LIN {X 0,Y 417.016,Z 627.534,A -85,B 0,C 180,E1 -10173.865,E2 -10173.865} C_VEL
LIN {X 0,Y 417.122,Z 624.59,A -85,B 0,C 180,E1 -10175.317,E2 -10175.317} C_VEL
LIN {X 0,Y 417.232,Z 620.603,A -85,B 0,C 180,E1 -10176.771,E2 -10176.771} C_VEL
LIN {X 0,Y 417.503,Z 614.475,A -85,B 0,C 180,E1 -10178.47,E2 -10178.47} C_VEL
LIN {X 0,Y 417.901,Z 607.782,A -85,B 0,C 180,E1 -10179.926,E2 -10179.926} C_VEL
LIN {X 0,Y 418.469,Z 599.483,A -85,B 0,C 180,E1 -10181.381,E2 -10181.381} C_VEL
LIN {X 0,Y 419.119,Z 590.981,A -85,B 0,C 180,E1 -10182.591,E2 -10182.591} C_VEL
LIN {X 0,Y 419.778,Z 581.378,A -85,B 0,C 180,E1 -10183.708,E2 -10183.708} C_VEL
LIN {X 0,Y 420.547,Z 570.086,A -85,B 0,C 180,E1 -10184.764,E2 -10184.764} C_VEL
LIN {X 0,Y 421.293,Z 558.7,A -85,B 0,C 180,E1 -10185.604,E2 -10185.604} C_VEL
LIN {X 0,Y 421.95,Z 547.015,A -85,B 0,C 180,E1 -10186.262,E2 -10186.262} C_VEL
LIN {X 0,Y 422.541,Z 534.469,A -85,B 0,C 180,E1 -10186.766,E2 -10186.766} C_VEL
LIN {X 0,Y 422.903,Z 521.748,A -85,B 0,C 180,E1 -10187.094,E2 -10187.094} C_VEL
LIN {X 0,Y 423.634,Z 443.257,A -85,B 0,C 180,E1 -10188.435,E2 -10188.435} C_VEL
LIN {X 0,Y 419.657,Z 417.924,A -85,B 0,C 180,E1 -10189.065,E2 -10189.065} C_VEL
LIN {X 0,Y 420.847,Z 399.93,A -85,B 0,C 180,E1 -10192.587,E2 -10192.587} C_VEL
LIN {X 0,Y 421.466,Z 390.877,A -85,B 0,C 180,E1 -10194.375,E2 -10194.375} C_VEL
LIN {X 0,Y 419.594,Z 380.403,A -85,B 0,C 180,E1 -10196.618,E2 -10196.618} C_VEL
LIN {X 0,Y 418.306,Z 374.38,A -85,B 0,C 180,E1 -10198.004,E2 -10198.004} C_VEL
LIN {X 0,Y 418.211,Z 374.394,A -85,B 0,C 180,E1 -10201.395,E2 -10201.395} C_VEL
LIN {X 0,Y 418.264,Z 374.38,A -85,B 0,C 180,E1 -10204.58,E2 -10204.58} C_VEL
LIN {X 0,Y 418.233,Z 374.389,A -85,B 0,C 180,E1 -10207.834,E2 -10207.834} C_VEL
LIN {X 0,Y 418.258,Z 374.382,A -85,B 0,C 180,E1 -10210.943,E2 -10210.943} C_VEL
LIN {X 0,Y 418.214,Z 374.392,A -85,B 0,C 180,E1 -10213.73,E2 -10213.73} C_VEL
LIN {X 0,Y 418.264,Z 374.38,A -85,B 0,C 180,E1 -10216.456,E2 -10216.456} C_VEL
LIN {X 0,Y 418.263,Z 374.383,A -85,B 0,C 180,E1 -10219.122,E2 -10219.122} C_VEL
LIN {X 0,Y 418.233,Z 374.385,A -85,B 0,C 180,E1 -10222.164,E2 -10222.164} C_VEL
LIN {X 0,Y 418.26,Z 374.388,A -85,B 0,C 180,E1 -10225.419,E2 -10225.419} C_VEL
LIN {X 0,Y 418.21,Z 374.387,A -85,B 0,C 180,E1 -10228.604,E2 -10228.604} C_VEL
LIN {X 0,Y 418.289,Z 374.378,A -85,B 0,C 180,E1 -10231.936,E2 -10231.936} C_VEL
LIN {X 0,Y 418.283,Z 374.384,A -85,B 0,C 180,E1 -10235.162,E2 -10235.162} C_VEL
LIN {X 0,Y 418.228,Z 374.385,A -85,B 0,C 180,E1 -10238.303,E2 -10238.303} C_VEL
LIN {X 0,Y 418.276,Z 374.384,A -85,B 0,C 180,E1 -10241.383,E2 -10241.383} C_VEL
LIN {X 0,Y 418.294,Z 374.377,A -85,B 0,C 180,E1 -10244.406,E2 -10244.406} C_VEL
LIN {X 0,Y 418.362,Z 374.372,A -85,B 0,C 180,E1 -10247.386,E2 -10247.386} C_VEL
LIN {X 0,Y 418.353,Z 374.369,A -85,B 0,C 180,E1 -10250.329,E2 -10250.329} C_VEL
LIN {X 0,Y 418.485,Z 374.357,A -85,B 0,C 180,E1 -10253.249,E2 -10253.249} C_VEL
LIN {X 0,Y 418.335,Z 374.376,A -85,B 0,C 180,E1 -10255.182,E2 -10255.182} C_VEL
LIN {X 0,Y 418.537,Z 374.346,A -85,B 0,C 180,E1 -10258.075,E2 -10258.075} C_VEL
LIN {X 0,Y 418.666,Z 374.33,A -85,B 0,C 180,E1 -10260,E2 -10260} C_VEL
LIN {X 0,Y 418.504,Z 374.358,A -85,B 0,C 180,E1 -10262.888,E2 -10262.888} C_VEL
LIN {X 0,Y 418.486,Z 374.359,A -85,B 0,C 180,E1 -10266.751,E2 -10266.751} C_VEL
LIN {X 0,Y 418.352,Z 374.369,A -85,B 0,C 180,E1 -10269.671,E2 -10269.671} C_VEL
LIN {X 0,Y 418.347,Z 374.374,A -85,B 0,C 180,E1 -10273.007,E2 -10273.007} C_VEL
LIN {X 0,Y 418.305,Z 374.382,A -85,B 0,C 180,E1 -10276.736,E2 -10276.736} C_VEL
LIN {X 0,Y 418.264,Z 374.38,A -85,B 0,C 180,E1 -10279.791,E2 -10279.791} C_VEL
LIN {X 0,Y 418.231,Z 374.39,A -85,B 0,C 180,E1 -10282.737,E2 -10282.737} C_VEL
LIN {X 0,Y 418.264,Z 374.381,A -85,B 0,C 180,E1 -10285.905,E2 -10285.905} C_VEL
LIN {X 0,Y 418.258,Z 374.382,A -85,B 0,C 180,E1 -10289.163,E2 -10289.163} C_VEL
LIN {X 0,Y 418.252,Z 374.385,A -85,B 0,C 180,E1 -10292.845,E2 -10292.845} C_VEL
LIN {X 0,Y 418.243,Z 374.387,A -85,B 0,C 180,E1 -10296.239,E2 -10296.239} C_VEL
LIN {X 0,Y 418.26,Z 374.381,A -85,B 0,C 180,E1 -10299.681,E2 -10299.681} C_VEL
LIN {X 0,Y 418.282,Z 374.385,A -85,B 0,C 180,E1 -10302.33,E2 -10302.33} C_VEL
LIN {X 0,Y 418.248,Z 374.382,A -85,B 0,C 180,E1 -10305.112,E2 -10305.112} C_VEL
LIN {X 0,Y 418.238,Z 374.385,A -85,B 0,C 180,E1 -10307.768,E2 -10307.768} C_VEL
LIN {X 0,Y 418.258,Z 374.384,A -85,B 0,C 180,E1 -10310.619,E2 -10310.619} C_VEL
LIN {X 0,Y 418.245,Z 374.387,A -85,B 0,C 180,E1 -10313.977,E2 -10313.977} C_VEL
LIN {X 0,Y 418.257,Z 374.381,A -85,B 0,C 180,E1 -10317.157,E2 -10317.157} C_VEL
LIN {X 0,Y 418.269,Z 374.38,A -85,B 0,C 180,E1 -10320.896,E2 -10320.896} C_VEL
LIN {X 0,Y 418.269,Z 374.387,A -85,B 0,C 180,E1 -10324.096,E2 -10324.096} C_VEL
LIN {X 0,Y 418.25,Z 374.479,A -85,B 0,C 180,E1 -10327.293,E2 -10327.293} C_VEL
LIN {X 0,Y 419.963,Z 383.206,A -85,B 0,C 180,E1 -10329.579,E2 -10329.579} C_VEL
LIN {X 0,Y 420.227,Z 386.742,A -85,B 0,C 180,E1 -10330.459,E2 -10330.459} C_VEL
LIN {X 0,Y 420.053,Z 389.099,A -85,B 0,C 180,E1 -10331.02,E2 -10331.02} C_VEL
LIN {X 0,Y 424.09,Z 408.927,A -85,B 0,C 180,E1 -10331.56,E2 -10331.56} C_VEL
LIN {X 0,Y 423.113,Z 496.309,A -85,B 0,C 180,E1 -10333.071,E2 -10333.071} C_VEL
LIN {X 0,Y 422.612,Z 510.138,A -85,B 0,C 180,E1 -10333.516,E2 -10333.516} C_VEL
LIN {X 0,Y 422.063,Z 522.517,A -85,B 0,C 180,E1 -10334.115,E2 -10334.115} C_VEL
LIN {X 0,Y 421.498,Z 534.349,A -85,B 0,C 180,E1 -10334.899,E2 -10334.899} C_VEL
LIN {X 0,Y 420.864,Z 544.797,A -85,B 0,C 180,E1 -10335.778,E2 -10335.778} C_VEL
LIN {X 0,Y 420.185,Z 554.863,A -85,B 0,C 180,E1 -10336.827,E2 -10336.827} C_VEL
LIN {X 0,Y 419.491,Z 563.403,A -85,B 0,C 180,E1 -10337.912,E2 -10337.912} C_VEL
LIN {X 0,Y 418.903,Z 571.264,A -85,B 0,C 180,E1 -10339.121,E2 -10339.121} C_VEL
LIN {X 0,Y 418.314,Z 578.947,A -85,B 0,C 180,E1 -10340.572,E2 -10340.572} C_VEL
LIN {X 0,Y 417.789,Z 585.995,A -85,B 0,C 180,E1 -10342.266,E2 -10342.266} C_VEL
LIN {X 0,Y 417.601,Z 589.304,A -85,B 0,C 180,E1 -10343.245,E2 -10343.245} C_VEL
LIN {X 0,Y 416.888,Z 591.511,A -85,B 0,C 180,E1 -10343.994,E2 -10343.994} C_VEL
LIN {X 0,Y 413.901,Z 594.609,A -85,B 0,C 180,E1 -10345.222,E2 -10345.222} C_VEL
LIN {X 0,Y 411.354,Z 596.611,A -85,B 0,C 180,E1 -10346.233,E2 -10346.233} C_VEL
LIN {X 0,Y 410.212,Z 597.769,A -85,B 0,C 180,E1 -10347.029,E2 -10347.029} C_VEL
LIN {X 0,Y 410.095,Z 598.052,A -85,B 0,C 180,E1 -10347.302,E2 -10347.302} C_VEL
LIN {X 0,Y 409.96,Z 599.41,A -85,B 0,C 180,E1 -10349.018,E2 -10349.018} C_VEL
LIN {X 0,Y 409.949,Z 599.643,A -85,B 0,C 180,E1 -10350,E2 -10350} C_VEL
LIN {X 0,Y 409.96,Z 599.455,A -85,B 0,C 180,E1 -10350.982,E2 -10350.982} C_VEL
LIN {X 0,Y 410.131,Z 597.905,A -85,B 0,C 180,E1 -10352.947,E2 -10352.947} C_VEL
LIN {X 0,Y 410.122,Z 596.556,A -85,B 0,C 180,E1 -10353.93,E2 -10353.93} C_VEL
LIN {X 0,Y 410.301,Z 593.697,A -85,B 0,C 180,E1 -10355.406,E2 -10355.406} C_VEL
LIN {X 0,Y 410.543,Z 589.82,A -85,B 0,C 180,E1 -10356.882,E2 -10356.882} C_VEL
LIN {X 0,Y 410.856,Z 584.818,A -85,B 0,C 180,E1 -10358.36,E2 -10358.36} C_VEL
LIN {X 0,Y 411.393,Z 578.516,A -85,B 0,C 180,E1 -10359.836,E2 -10359.836} C_VEL
LIN {X 0,Y 412.034,Z 570.627,A -85,B 0,C 180,E1 -10361.312,E2 -10361.312} C_VEL
LIN {X 0,Y 412.639,Z 562.584,A -85,B 0,C 180,E1 -10362.542,E2 -10362.542} C_VEL
LIN {X 0,Y 413.512,Z 552.76,A -85,B 0,C 180,E1 -10363.765,E2 -10363.765} C_VEL
LIN {X 0,Y 414.125,Z 543.099,A -85,B 0,C 180,E1 -10364.747,E2 -10364.747} C_VEL
LIN {X 0,Y 414.814,Z 532.639,A -85,B 0,C 180,E1 -10365.602,E2 -10365.602} C_VEL
LIN {X 0,Y 415.467,Z 520.04,A -85,B 0,C 180,E1 -10366.396,E2 -10366.396} C_VEL
LIN {X 0,Y 416.011,Z 507.426,A -85,B 0,C 180,E1 -10366.974,E2 -10366.974} C_VEL
LIN {X 0,Y 416.372,Z 495.481,A -85,B 0,C 180,E1 -10367.338,E2 -10367.338} C_VEL
LIN {X 0,Y 417.31,Z 409.13,A -85,B 0,C 180,E1 -10368.85,E2 -10368.85} C_VEL
LIN {X 0,Y 413.176,Z 389.255,A -85,B 0,C 180,E1 -10369.436,E2 -10369.436} C_VEL
LIN {X 0,Y 413.003,Z 384.502,A -85,B 0,C 180,E1 -10370.621,E2 -10370.621} C_VEL
LIN {X 0,Y 411.231,Z 375.268,A -85,B 0,C 180,E1 -10373.11,E2 -10373.11} C_VEL
LIN {X 0,Y 411.239,Z 375.258,A -85,B 0,C 180,E1 -10376.38,E2 -10376.38} C_VEL
LIN {X 0,Y 411.2,Z 375.264,A -85,B 0,C 180,E1 -10379.712,E2 -10379.712} C_VEL
LIN {X 0,Y 411.206,Z 375.26,A -85,B 0,C 180,E1 -10383.155,E2 -10383.155} C_VEL
LIN {X 0,Y 411.194,Z 375.261,A -85,B 0,C 180,E1 -10386.552,E2 -10386.552} C_VEL
LIN {X 0,Y 411.216,Z 375.264,A -85,B 0,C 180,E1 -10389.728,E2 -10389.728} C_VEL
LIN {X 0,Y 411.171,Z 375.265,A -85,B 0,C 180,E1 -10393.133,E2 -10393.133} C_VEL
LIN {X 0,Y 411.224,Z 375.263,A -85,B 0,C 180,E1 -10395.872,E2 -10395.872} C_VEL
LIN {X 0,Y 411.206,Z 375.259,A -85,B 0,C 180,E1 -10398.763,E2 -10398.763} C_VEL
LIN {X 0,Y 411.199,Z 375.263,A -85,B 0,C 180,E1 -10402.027,E2 -10402.027} C_VEL
LIN {X 0,Y 411.201,Z 375.266,A -85,B 0,C 180,E1 -10405.666,E2 -10405.666} C_VEL
LIN {X 0,Y 411.183,Z 375.265,A -85,B 0,C 180,E1 -10409.152,E2 -10409.152} C_VEL
LIN {X 0,Y 411.252,Z 375.253,A -85,B 0,C 180,E1 -10412.522,E2 -10412.522} C_VEL
LIN {X 0,Y 411.221,Z 375.261,A -85,B 0,C 180,E1 -10415.784,E2 -10415.784} C_VEL
LIN {X 0,Y 411.191,Z 375.264,A -85,B 0,C 180,E1 -10418.965,E2 -10418.965} C_VEL
LIN {X 0,Y 411.245,Z 375.255,A -85,B 0,C 180,E1 -10422.084,E2 -10422.084} C_VEL
LIN {X 0,Y 411.255,Z 375.258,A -85,B 0,C 180,E1 -10425.147,E2 -10425.147} C_VEL
LIN {X 0,Y 411.291,Z 375.249,A -85,B 0,C 180,E1 -10428.167,E2 -10428.167} C_VEL
LIN {X 0,Y 411.474,Z 375.226,A -85,B 0,C 180,E1 -10432.146,E2 -10432.146} C_VEL
LIN {X 0,Y 411.467,Z 375.227,A -85,B 0,C 180,E1 -10434.118,E2 -10434.118} C_VEL
LIN {X 0,Y 411.506,Z 375.222,A -85,B 0,C 180,E1 -10438.042,E2 -10438.042} C_VEL
LIN {X 0,Y 411.635,Z 375.206,A -85,B 0,C 180,E1 -10440,E2 -10440} C_VEL
LIN {X 0,Y 411.46,Z 375.233,A -85,B 0,C 180,E1 -10442.937,E2 -10442.937} C_VEL
LIN {X 0,Y 411.453,Z 375.234,A -85,B 0,C 180,E1 -10446.867,E2 -10446.867} C_VEL
LIN {X 0,Y 411.301,Z 375.247,A -85,B 0,C 180,E1 -10449.839,E2 -10449.839} C_VEL
LIN {X 0,Y 411.305,Z 375.252,A -85,B 0,C 180,E1 -10453.109,E2 -10453.109} C_VEL
LIN {X 0,Y 411.249,Z 375.261,A -85,B 0,C 180,E1 -10456.889,E2 -10456.889} C_VEL
LIN {X 0,Y 411.223,Z 375.257,A -85,B 0,C 180,E1 -10459.987,E2 -10459.987} C_VEL
LIN {X 0,Y 411.196,Z 375.263,A -85,B 0,C 180,E1 -10463.148,E2 -10463.148} C_VEL
LIN {X 0,Y 411.231,Z 375.259,A -85,B 0,C 180,E1 -10466.381,E2 -10466.381} C_VEL
LIN {X 0,Y 411.194,Z 375.261,A -85,B 0,C 180,E1 -10469.713,E2 -10469.713} C_VEL
LIN {X 0,Y 411.2,Z 375.262,A -85,B 0,C 180,E1 -10473.156,E2 -10473.156} C_VEL
LIN {X 0,Y 411.19,Z 375.268,A -85,B 0,C 180,E1 -10476.554,E2 -10476.554} C_VEL
LIN {X 0,Y 411.223,Z 375.257,A -85,B 0,C 180,E1 -10479.731,E2 -10479.731} C_VEL
LIN {X 0,Y 411.218,Z 375.259,A -85,B 0,C 180,E1 -10483.128,E2 -10483.128} C_VEL
LIN {X 0,Y 411.173,Z 375.265,A -85,B 0,C 180,E1 -10485.88,E2 -10485.88} C_VEL
LIN {X 0,Y 411.203,Z 375.26,A -85,B 0,C 180,E1 -10489.5,E2 -10489.5} C_VEL
LIN {X 0,Y 411.199,Z 375.263,A -85,B 0,C 180,E1 -10492.028,E2 -10492.028} C_VEL
LIN {X 0,Y 411.205,Z 375.26,A -85,B 0,C 180,E1 -10495.667,E2 -10495.667} C_VEL
LIN {X 0,Y 411.19,Z 375.264,A -85,B 0,C 180,E1 -10499.153,E2 -10499.153} C_VEL
LIN {X 0,Y 411.253,Z 375.293,A -85,B 0,C 180,E1 -10501.762,E2 -10501.762} C_VEL
LIN {X 0,Y 413.552,Z 386.393,A -85,B 0,C 180,E1 -10504.25,E2 -10504.25} C_VEL
LIN {X 0,Y 414.502,Z 391.964,A -85,B 0,C 180,E1 -10505.456,E2 -10505.456} C_VEL
LIN {X 0,Y 413.807,Z 402.306,A -85,B 0,C 180,E1 -10507.535,E2 -10507.535} C_VEL
LIN {X 0,Y 412.779,Z 417.545,A -85,B 0,C 180,E1 -10510.578,E2 -10510.578} C_VEL
LIN {X 0,Y 417.006,Z 444.934,A -85,B 0,C 180,E1 -10511.29,E2 -10511.29} C_VEL
LIN {X 0,Y 416.056,Z 526.083,A -85,B 0,C 180,E1 -10512.711,E2 -10512.711} C_VEL
LIN {X 0,Y 415.527,Z 539.325,A -85,B 0,C 180,E1 -10513.132,E2 -10513.132} C_VEL
LIN {X 0,Y 414.9,Z 551.477,A -85,B 0,C 180,E1 -10513.707,E2 -10513.707} C_VEL
LIN {X 0,Y 414.074,Z 563.741,A -85,B 0,C 180,E1 -10514.495,E2 -10514.495} C_VEL
LIN {X 0,Y 413.229,Z 575.345,A -85,B 0,C 180,E1 -10515.472,E2 -10515.472} C_VEL
LIN {X 0,Y 412.501,Z 585.795,A -85,B 0,C 180,E1 -10516.577,E2 -10516.577} C_VEL
LIN {X 0,Y 411.898,Z 594.345,A -85,B 0,C 180,E1 -10517.686,E2 -10517.686} C_VEL
LIN {X 0,Y 411.256,Z 602.232,A -85,B 0,C 180,E1 -10518.916,E2 -10518.916} C_VEL
LIN {X 0,Y 410.702,Z 609.941,A -85,B 0,C 180,E1 -10520.396,E2 -10520.396} C_VEL
LIN {X 0,Y 410.288,Z 617.052,A -85,B 0,C 180,E1 -10522.124,E2 -10522.124} C_VEL
LIN {X 0,Y 410.043,Z 622.276,A -85,B 0,C 180,E1 -10523.775,E2 -10523.775} C_VEL
LIN {X 0,Y 410.019,Z 625.406,A -85,B 0,C 180,E1 -10525.084,E2 -10525.084} C_VEL
LIN {X 0,Y 409.934,Z 627.271,A -85,B 0,C 180,E1 -10526.068,E2 -10526.068} C_VEL
LIN {X 0,Y 409.997,Z 629.673,A -85,B 0,C 180,E1 -10528.035,E2 -10528.035} C_VEL
LIN {X 0,Y 409.956,Z 630.282,A -85,B 0,C 180,E1 -10529.018,E2 -10529.018} C_VEL
LIN {X 0,Y 409.948,Z 630.498,A -85,B 0,C 180,E1 -10530,E2 -10530} C_VEL
LIN {X 0,Y 409.997,Z 629.671,A -85,B 0,C 180,E1 -10531.965,E2 -10531.965} C_VEL
LIN {X 0,Y 409.934,Z 627.266,A -85,B 0,C 180,E1 -10533.932,E2 -10533.932} C_VEL
LIN {X 0,Y 410.018,Z 624.32,A -85,B 0,C 180,E1 -10535.409,E2 -10535.409} C_VEL
LIN {X 0,Y 410.164,Z 620.334,A -85,B 0,C 180,E1 -10536.889,E2 -10536.889} C_VEL
LIN {X 0,Y 410.465,Z 614.205,A -85,B 0,C 180,E1 -10538.616,E2 -10538.616} C_VEL
LIN {X 0,Y 410.881,Z 607.512,A -85,B 0,C 180,E1 -10540.097,E2 -10540.097} C_VEL
LIN {X 0,Y 411.488,Z 599.213,A -85,B 0,C 180,E1 -10541.577,E2 -10541.577} C_VEL
LIN {X 0,Y 412.143,Z 590.709,A -85,B 0,C 180,E1 -10542.807,E2 -10542.807} C_VEL
LIN {X 0,Y 412.883,Z 580.441,A -85,B 0,C 180,E1 -10544.012,E2 -10544.012} C_VEL
LIN {X 0,Y 413.671,Z 569.815,A -85,B 0,C 180,E1 -10545.016,E2 -10545.016} C_VEL
LIN {X 0,Y 414.448,Z 558.428,A -85,B 0,C 180,E1 -10545.869,E2 -10545.869} C_VEL
LIN {X 0,Y 415.135,Z 546.741,A -85,B 0,C 180,E1 -10546.536,E2 -10546.536} C_VEL
LIN {X 0,Y 415.797,Z 533.277,A -85,B 0,C 180,E1 -10547.078,E2 -10547.078} C_VEL
LIN {X 0,Y 416.165,Z 519.934,A -85,B 0,C 180,E1 -10547.411,E2 -10547.411} C_VEL
LIN {X 0,Y 416.873,Z 443.749,A -85,B 0,C 180,E1 -10548.731,E2 -10548.731} C_VEL
LIN {X 0,Y 412.774,Z 417.524,A -85,B 0,C 180,E1 -10549.422,E2 -10549.422} C_VEL
LIN {X 0,Y 414.009,Z 399.679,A -85,B 0,C 180,E1 -10552.981,E2 -10552.981} C_VEL
LIN {X 0,Y 414.518,Z 391.925,A -85,B 0,C 180,E1 -10554.543,E2 -10554.543} C_VEL
LIN {X 0,Y 412.32,Z 380.147,A -85,B 0,C 180,E1 -10557.126,E2 -10557.126} C_VEL
LIN {X 0,Y 411.25,Z 375.26,A -85,B 0,C 180,E1 -10558.239,E2 -10558.239} C_VEL
LIN {X 0,Y 411.165,Z 375.272,A -85,B 0,C 180,E1 -10561.996,E2 -10561.996} C_VEL
LIN {X 0,Y 411.21,Z 375.259,A -85,B 0,C 180,E1 -10564.878,E2 -10564.878} C_VEL
LIN {X 0,Y 411.209,Z 375.261,A -85,B 0,C 180,E1 -10568.169,E2 -10568.169} C_VEL
LIN {X 0,Y 411.191,Z 375.264,A -85,B 0,C 180,E1 -10571.232,E2 -10571.232} C_VEL
LIN {X 0,Y 411.185,Z 375.262,A -85,B 0,C 180,E1 -10574.488,E2 -10574.488} C_VEL
LIN {X 0,Y 411.225,Z 375.261,A -85,B 0,C 180,E1 -10577.296,E2 -10577.296} C_VEL
LIN {X 0,Y 411.226,Z 375.257,A -85,B 0,C 180,E1 -10580.777,E2 -10580.777} C_VEL
LIN {X 0,Y 411.194,Z 375.261,A -85,B 0,C 180,E1 -10584.471,E2 -10584.471} C_VEL
LIN {X 0,Y 411.201,Z 375.262,A -85,B 0,C 180,E1 -10586.873,E2 -10586.873} C_VEL
LIN {X 0,Y 411.234,Z 375.256,A -85,B 0,C 180,E1 -10590.642,E2 -10590.642} C_VEL
LIN {X 0,Y 411.231,Z 375.26,A -85,B 0,C 180,E1 -10593.619,E2 -10593.619} C_VEL
LIN {X 0,Y 411.196,Z 375.263,A -85,B 0,C 180,E1 -10596.852,E2 -10596.852} C_VEL
LIN {X 0,Y 411.208,Z 375.259,A -85,B 0,C 180,E1 -10600.05,E2 -10600.05} C_VEL
LIN {X 0,Y 411.255,Z 375.26,A -85,B 0,C 180,E1 -10603.131,E2 -10603.131} C_VEL
LIN {X 0,Y 411.305,Z 375.251,A -85,B 0,C 180,E1 -10606.891,E2 -10606.891} C_VEL
LIN {X 0,Y 411.301,Z 375.247,A -85,B 0,C 180,E1 -10610.161,E2 -10610.161} C_VEL
LIN {X 0,Y 411.452,Z 375.235,A -85,B 0,C 180,E1 -10613.133,E2 -10613.133} C_VEL
LIN {X 0,Y 411.305,Z 375.253,A -85,B 0,C 180,E1 -10615.099,E2 -10615.099} C_VEL
LIN {X 0,Y 411.506,Z 375.222,A -85,B 0,C 180,E1 -10618.043,E2 -10618.043} C_VEL
LIN {X 0,Y 411.635,Z 375.206,A -85,B 0,C 180,E1 -10620,E2 -10620} C_VEL
LIN {X 0,Y 411.46,Z 375.235,A -85,B 0,C 180,E1 -10622.937,E2 -10622.937} C_VEL
LIN {X 0,Y 411.453,Z 375.236,A -85,B 0,C 180,E1 -10626.867,E2 -10626.867} C_VEL
LIN {X 0,Y 411.301,Z 375.247,A -85,B 0,C 180,E1 -10629.839,E2 -10629.839} C_VEL
LIN {X 0,Y 411.305,Z 375.25,A -85,B 0,C 180,E1 -10633.109,E2 -10633.109} C_VEL
LIN {X 0,Y 411.25,Z 375.259,A -85,B 0,C 180,E1 -10636.889,E2 -10636.889} C_VEL
LIN {X 0,Y 411.223,Z 375.258,A -85,B 0,C 180,E1 -10639.987,E2 -10639.987} C_VEL
LIN {X 0,Y 411.197,Z 375.262,A -85,B 0,C 180,E1 -10643.148,E2 -10643.148} C_VEL
LIN {X 0,Y 411.231,Z 375.261,A -85,B 0,C 180,E1 -10646.382,E2 -10646.382} C_VEL
LIN {X 0,Y 411.194,Z 375.261,A -85,B 0,C 180,E1 -10649.713,E2 -10649.713} C_VEL
LIN {X 0,Y 411.201,Z 375.261,A -85,B 0,C 180,E1 -10653.157,E2 -10653.157} C_VEL
LIN {X 0,Y 411.191,Z 375.267,A -85,B 0,C 180,E1 -10656.554,E2 -10656.554} C_VEL
LIN {X 0,Y 411.223,Z 375.258,A -85,B 0,C 180,E1 -10659.731,E2 -10659.731} C_VEL
LIN {X 0,Y 411.218,Z 375.258,A -85,B 0,C 180,E1 -10663.128,E2 -10663.128} C_VEL
LIN {X 0,Y 411.17,Z 375.266,A -85,B 0,C 180,E1 -10665.881,E2 -10665.881} C_VEL
LIN {X 0,Y 411.162,Z 375.267,A -85,B 0,C 180,E1 -10668.772,E2 -10668.772} C_VEL
LIN {X 0,Y 411.21,Z 375.262,A -85,B 0,C 180,E1 -10671.831,E2 -10671.831} C_VEL
LIN {X 0,Y 411.21,Z 375.259,A -85,B 0,C 180,E1 -10675.122,E2 -10675.122} C_VEL
LIN {X 0,Y 411.165,Z 375.27,A -85,B 0,C 180,E1 -10678.004,E2 -10678.004} C_VEL
LIN {X 0,Y 411.218,Z 375.258,A -85,B 0,C 180,E1 -10681.411,E2 -10681.411} C_VEL
LIN {X 0,Y 411.237,Z 375.258,A -85,B 0,C 180,E1 -10683.62,E2 -10683.62} C_VEL
LIN {X 0,Y 411.221,Z 375.325,A -85,B 0,C 180,E1 -10687.039,E2 -10687.039} C_VEL
LIN {X 0,Y 413.161,Z 385.572,A -85,B 0,C 180,E1 -10689.757,E2 -10689.757} C_VEL
LIN {X 0,Y 413.182,Z 389.279,A -85,B 0,C 180,E1 -10690.672,E2 -10690.672} C_VEL
LIN {X 0,Y 417.36,Z 409.465,A -85,B 0,C 180,E1 -10691.256,E2 -10691.256} C_VEL
LIN {X 0,Y 416.332,Z 496.593,A -85,B 0,C 180,E1 -10692.786,E2 -10692.786} C_VEL
LIN {X 0,Y 415.82,Z 510.416,A -85,B 0,C 180,E1 -10693.239,E2 -10693.239} C_VEL
LIN {X 0,Y 415.259,Z 522.791,A -85,B 0,C 180,E1 -10693.848,E2 -10693.848} C_VEL
LIN {X 0,Y 414.645,Z 534.622,A -85,B 0,C 180,E1 -10694.643,E2 -10694.643} C_VEL
LIN {X 0,Y 413.942,Z 545.731,A -85,B 0,C 180,E1 -10695.6,E2 -10695.6} C_VEL
LIN {X 0,Y 413.207,Z 556.192,A -85,B 0,C 180,E1 -10696.726,E2 -10696.726} C_VEL
LIN {X 0,Y 412.445,Z 565.365,A -85,B 0,C 180,E1 -10697.952,E2 -10697.952} C_VEL
LIN {X 0,Y 411.709,Z 574.268,A -85,B 0,C 180,E1 -10699.426,E2 -10699.426} C_VEL
LIN {X 0,Y 411.127,Z 581.433,A -85,B 0,C 180,E1 -10700.902,E2 -10700.902} C_VEL
LIN {X 0,Y 410.742,Z 586.264,A -85,B 0,C 180,E1 -10702.133,E2 -10702.133} C_VEL
LIN {X 0,Y 410.528,Z 590.635,A -85,B 0,C 180,E1 -10703.5,E2 -10703.5} C_VEL
LIN {X 0,Y 410.194,Z 594.55,A -85,B 0,C 180,E1 -10705.086,E2 -10705.086} C_VEL
LIN {X 0,Y 410.124,Z 596.405,A -85,B 0,C 180,E1 -10706.07,E2 -10706.07} C_VEL
LIN {X 0,Y 410.095,Z 598.052,A -85,B 0,C 180,E1 -10707.302,E2 -10707.302} C_VEL
LIN {X 0,Y 409.34,Z 598.905,A -85,B 0,C 180,E1 -10708.114,E2 -10708.114} C_VEL
LIN {X 0,Y 406.39,Z 599.689,A -85,B 0,C 180,E1 -10709.441,E2 -10709.441} C_VEL
LIN {X 0,Y 403.971,Z 599.802,A -85,B 0,C 180,E1 -10710.515,E2 -10710.515} C_VEL
LIN {X 0,Y 402.979,Z 599.554,A -85,B 0,C 180,E1 -10711.345,E2 -10711.345} C_VEL
LIN {X 0,Y 402.922,Z 599.355,A -85,B 0,C 180,E1 -10711.625,E2 -10711.625} C_VEL
LIN {X 0,Y 403.051,Z 598.171,A -85,B 0,C 180,E1 -10712.999,E2 -10712.999} C_VEL
LIN {X 0,Y 403.034,Z 596.823,A -85,B 0,C 180,E1 -10714,E2 -10714} C_VEL
LIN {X 0,Y 403.254,Z 593.962,A -85,B 0,C 180,E1 -10715.5,E2 -10715.5} C_VEL
LIN {X 0,Y 403.489,Z 590.086,A -85,B 0,C 180,E1 -10717.003,E2 -10717.003} C_VEL
LIN {X 0,Y 403.842,Z 585.083,A -85,B 0,C 180,E1 -10718.506,E2 -10718.506} C_VEL
LIN {X 0,Y 404.4,Z 578.781,A -85,B 0,C 180,E1 -10720.008,E2 -10720.008} C_VEL
LIN {X 0,Y 405.082,Z 570.891,A -85,B 0,C 180,E1 -10721.509,E2 -10721.509} C_VEL
LIN {X 0,Y 405.721,Z 562.848,A -85,B 0,C 180,E1 -10722.759,E2 -10722.759} C_VEL
LIN {X 0,Y 406.628,Z 553.023,A -85,B 0,C 180,E1 -10724.003,E2 -10724.003} C_VEL
LIN {X 0,Y 407.328,Z 541.979,A -85,B 0,C 180,E1 -10725.127,E2 -10725.127} C_VEL
LIN {X 0,Y 408.092,Z 531.142,A -85,B 0,C 180,E1 -10725.994,E2 -10725.994} C_VEL
LIN {X 0,Y 408.762,Z 519.17,A -85,B 0,C 180,E1 -10726.737,E2 -10726.737} C_VEL
LIN {X 0,Y 409.253,Z 506.9,A -85,B 0,C 180,E1 -10727.295,E2 -10727.295} C_VEL
LIN {X 0,Y 409.604,Z 494.262,A -85,B 0,C 180,E1 -10727.666,E2 -10727.666} C_VEL
LIN {X 0,Y 410.593,Z 410.055,A -85,B 0,C 180,E1 -10729.157,E2 -10729.157} C_VEL
LIN {X 0,Y 406.271,Z 389.627,A -85,B 0,C 180,E1 -10729.753,E2 -10729.753} C_VEL
LIN {X 0,Y 405.974,Z 385.524,A -85,B 0,C 180,E1 -10730.8,E2 -10730.8} C_VEL
LIN {X 0,Y 404.198,Z 376.144,A -85,B 0,C 180,E1 -10733.375,E2 -10733.375} C_VEL
LIN {X 0,Y 404.184,Z 376.14,A -85,B 0,C 180,E1 -10735.766,E2 -10735.766} C_VEL
LIN {X 0,Y 404.195,Z 376.14,A -85,B 0,C 180,E1 -10737.999,E2 -10737.999} C_VEL
LIN {X 0,Y 404.139,Z 376.143,A -85,B 0,C 180,E1 -10741.557,E2 -10741.557} C_VEL
LIN {X 0,Y 404.184,Z 376.134,A -85,B 0,C 180,E1 -10745.015,E2 -10745.015} C_VEL
LIN {X 0,Y 404.157,Z 376.137,A -85,B 0,C 180,E1 -10748.756,E2 -10748.756} C_VEL
LIN {X 0,Y 404.121,Z 376.147,A -85,B 0,C 180,E1 -10751.599,E2 -10751.599} C_VEL
LIN {X 0,Y 404.152,Z 376.138,A -85,B 0,C 180,E1 -10754.523,E2 -10754.523} C_VEL
LIN {X 0,Y 404.203,Z 376.134,A -85,B 0,C 180,E1 -10757.304,E2 -10757.304} C_VEL
LIN {X 0,Y 404.165,Z 376.14,A -85,B 0,C 180,E1 -10759.955,E2 -10759.955} C_VEL
LIN {X 0,Y 404.136,Z 376.142,A -85,B 0,C 180,E1 -10763.123,E2 -10763.123} C_VEL
LIN {X 0,Y 404.14,Z 376.141,A -85,B 0,C 180,E1 -10766.187,E2 -10766.187} C_VEL
LIN {X 0,Y 404.139,Z 376.145,A -85,B 0,C 180,E1 -10769.714,E2 -10769.714} C_VEL
LIN {X 0,Y 404.189,Z 376.136,A -85,B 0,C 180,E1 -10773.122,E2 -10773.122} C_VEL
LIN {X 0,Y 404.171,Z 376.141,A -85,B 0,C 180,E1 -10775.334,E2 -10775.334} C_VEL
LIN {X 0,Y 404.133,Z 376.141,A -85,B 0,C 180,E1 -10778.58,E2 -10778.58} C_VEL
LIN {X 0,Y 404.203,Z 376.134,A -85,B 0,C 180,E1 -10781.761,E2 -10781.761} C_VEL
LIN {X 0,Y 404.2,Z 376.134,A -85,B 0,C 180,E1 -10784.882,E2 -10784.882} C_VEL
LIN {X 0,Y 404.262,Z 376.125,A -85,B 0,C 180,E1 -10787.959,E2 -10787.959} C_VEL
LIN {X 0,Y 404.425,Z 376.104,A -85,B 0,C 180,E1 -10792.099,E2 -10792.099} C_VEL
LIN {X 0,Y 404.416,Z 376.105,A -85,B 0,C 180,E1 -10794.015,E2 -10794.015} C_VEL
LIN {X 0,Y 404.475,Z 376.098,A -85,B 0,C 180,E1 -10798.008,E2 -10798.008} C_VEL
LIN {X 0,Y 404.605,Z 376.082,A -85,B 0,C 180,E1 -10800,E2 -10800} C_VEL
LIN {X 0,Y 404.417,Z 376.111,A -85,B 0,C 180,E1 -10802.988,E2 -10802.988} C_VEL
LIN {X 0,Y 404.404,Z 376.114,A -85,B 0,C 180,E1 -10806.987,E2 -10806.987} C_VEL
LIN {X 0,Y 404.264,Z 376.124,A -85,B 0,C 180,E1 -10810.012,E2 -10810.012} C_VEL
LIN {X 0,Y 404.258,Z 376.128,A -85,B 0,C 180,E1 -10813.212,E2 -10813.212} C_VEL
LIN {X 0,Y 404.208,Z 376.136,A -85,B 0,C 180,E1 -10817.007,E2 -10817.007} C_VEL
LIN {X 0,Y 404.157,Z 376.14,A -85,B 0,C 180,E1 -10820.352,E2 -10820.352} C_VEL
LIN {X 0,Y 404.163,Z 376.137,A -85,B 0,C 180,E1 -10823.575,E2 -10823.575} C_VEL
LIN {X 0,Y 404.177,Z 376.135,A -85,B 0,C 180,E1 -10825.767,E2 -10825.767} C_VEL
LIN {X 0,Y 404.189,Z 376.134,A -85,B 0,C 180,E1 -10828,E2 -10828} C_VEL
LIN {X 0,Y 404.133,Z 376.14,A -85,B 0,C 180,E1 -10831.559,E2 -10831.559} C_VEL
LIN {X 0,Y 404.18,Z 376.137,A -85,B 0,C 180,E1 -10835.017,E2 -10835.017} C_VEL
LIN {X 0,Y 404.159,Z 376.142,A -85,B 0,C 180,E1 -10838.757,E2 -10838.757} C_VEL
LIN {X 0,Y 404.187,Z 376.134,A -85,B 0,C 180,E1 -10841.611,E2 -10841.611} C_VEL
LIN {X 0,Y 404.186,Z 376.14,A -85,B 0,C 180,E1 -10844.529,E2 -10844.529} C_VEL
LIN {X 0,Y 404.136,Z 376.14,A -85,B 0,C 180,E1 -10847.297,E2 -10847.297} C_VEL
LIN {X 0,Y 404.166,Z 376.139,A -85,B 0,C 180,E1 -10849.956,E2 -10849.956} C_VEL
LIN {X 0,Y 404.138,Z 376.14,A -85,B 0,C 180,E1 -10853.125,E2 -10853.125} C_VEL
LIN {X 0,Y 404.144,Z 376.145,A -85,B 0,C 180,E1 -10856.189,E2 -10856.189} C_VEL
LIN {X 0,Y 404.145,Z 376.141,A -85,B 0,C 180,E1 -10859.716,E2 -10859.716} C_VEL
LIN {X 0,Y 404.195,Z 376.192,A -85,B 0,C 180,E1 -10861.471,E2 -10861.471} C_VEL
LIN {X 0,Y 406.555,Z 387.292,A -85,B 0,C 180,E1 -10864.015,E2 -10864.015} C_VEL
LIN {X 0,Y 407.61,Z 394.313,A -85,B 0,C 180,E1 -10865.556,E2 -10865.556} C_VEL
LIN {X 0,Y 406.208,Z 411.786,A -85,B 0,C 180,E1 -10869.113,E2 -10869.113} C_VEL
LIN {X 0,Y 405.843,Z 417.359,A -85,B 0,C 180,E1 -10870.249,E2 -10870.249} C_VEL
LIN {X 0,Y 410.3,Z 445.803,A -85,B 0,C 180,E1 -10870.992,E2 -10870.992} C_VEL
LIN {X 0,Y 409.288,Z 525.828,A -85,B 0,C 180,E1 -10872.416,E2 -10872.416} C_VEL
LIN {X 0,Y 408.741,Z 539.066,A -85,B 0,C 180,E1 -10872.844,E2 -10872.844} C_VEL
LIN {X 0,Y 408.092,Z 551.216,A -85,B 0,C 180,E1 -10873.428,E2 -10873.428} C_VEL
LIN {X 0,Y 407.226,Z 563.477,A -85,B 0,C 180,E1 -10874.228,E2 -10874.228} C_VEL
LIN {X 0,Y 406.303,Z 575.336,A -85,B 0,C 180,E1 -10875.244,E2 -10875.244} C_VEL
LIN {X 0,Y 405.58,Z 585.305,A -85,B 0,C 180,E1 -10876.317,E2 -10876.317} C_VEL
LIN {X 0,Y 404.936,Z 594.079,A -85,B 0,C 180,E1 -10877.47,E2 -10877.47} C_VEL
LIN {X 0,Y 404.233,Z 601.965,A -85,B 0,C 180,E1 -10878.721,E2 -10878.721} C_VEL
LIN {X 0,Y 403.659,Z 609.673,A -85,B 0,C 180,E1 -10880.227,E2 -10880.227} C_VEL
LIN {X 0,Y 403.219,Z 616.785,A -85,B 0,C 180,E1 -10881.985,E2 -10881.985} C_VEL
LIN {X 0,Y 403.004,Z 621.52,A -85,B 0,C 180,E1 -10883.492,E2 -10883.492} C_VEL
LIN {X 0,Y 402.93,Z 625.139,A -85,B 0,C 180,E1 -10884.997,E2 -10884.997} C_VEL
LIN {X 0,Y 402.854,Z 627.004,A -85,B 0,C 180,E1 -10885.999,E2 -10885.999} C_VEL
LIN {X 0,Y 402.907,Z 629.407,A -85,B 0,C 180,E1 -10888.001,E2 -10888.001} C_VEL
LIN {X 0,Y 402.882,Z 630.016,A -85,B 0,C 180,E1 -10889,E2 -10889} C_VEL
LIN {X 0,Y 402.871,Z 630.231,A -85,B 0,C 180,E1 -10890,E2 -10890} C_VEL
LIN {X 0,Y 402.882,Z 630.013,A -85,B 0,C 180,E1 -10891,E2 -10891} C_VEL
LIN {X 0,Y 402.907,Z 629.404,A -85,B 0,C 180,E1 -10891.999,E2 -10891.999} C_VEL
LIN {X 0,Y 402.854,Z 626.999,A -85,B 0,C 180,E1 -10894.001,E2 -10894.001} C_VEL
LIN {X 0,Y 402.915,Z 624.051,A -85,B 0,C 180,E1 -10895.505,E2 -10895.505} C_VEL
LIN {X 0,Y 403.077,Z 620.064,A -85,B 0,C 180,E1 -10897.01,E2 -10897.01} C_VEL
LIN {X 0,Y 403.406,Z 613.935,A -85,B 0,C 180,E1 -10898.768,E2 -10898.768} C_VEL
LIN {X 0,Y 403.853,Z 607.242,A -85,B 0,C 180,E1 -10900.275,E2 -10900.275} C_VEL
LIN {X 0,Y 404.513,Z 598.943,A -85,B 0,C 180,E1 -10901.779,E2 -10901.779} C_VEL
LIN {X 0,Y 405.172,Z 590.437,A -85,B 0,C 180,E1 -10903.032,E2 -10903.032} C_VEL
LIN {X 0,Y 405.975,Z 580.169,A -85,B 0,C 180,E1 -10904.255,E2 -10904.255} C_VEL
LIN {X 0,Y 406.794,Z 569.543,A -85,B 0,C 180,E1 -10905.276,E2 -10905.276} C_VEL
LIN {X 0,Y 407.601,Z 558.155,A -85,B 0,C 180,E1 -10906.142,E2 -10906.142} C_VEL
LIN {X 0,Y 408.32,Z 546.466,A -85,B 0,C 180,E1 -10906.82,E2 -10906.82} C_VEL
LIN {X 0,Y 409.007,Z 532.999,A -85,B 0,C 180,E1 -10907.37,E2 -10907.37} C_VEL
LIN {X 0,Y 409.402,Z 519.649,A -85,B 0,C 180,E1 -10907.708,E2 -10907.708} C_VEL
LIN {X 0,Y 410.169,Z 444.803,A -85,B 0,C 180,E1 -10909.024,E2 -10909.024} C_VEL
LIN {X 0,Y 405.836,Z 417.414,A -85,B 0,C 180,E1 -10909.735,E2 -10909.735} C_VEL
LIN {X 0,Y 407.085,Z 400.713,A -85,B 0,C 180,E1 -10913.126,E2 -10913.126} C_VEL
LIN {X 0,Y 407.565,Z 392.966,A -85,B 0,C 180,E1 -10914.718,E2 -10914.718} C_VEL
LIN {X 0,Y 405.357,Z 381.426,A -85,B 0,C 180,E1 -10917.303,E2 -10917.303} C_VEL
LIN {X 0,Y 404.202,Z 376.138,A -85,B 0,C 180,E1 -10918.564,E2 -10918.564} C_VEL
LIN {X 0,Y 404.138,Z 376.147,A -85,B 0,C 180,E1 -10921.557,E2 -10921.557} C_VEL
LIN {X 0,Y 404.184,Z 376.135,A -85,B 0,C 180,E1 -10925.015,E2 -10925.015} C_VEL
LIN {X 0,Y 404.157,Z 376.138,A -85,B 0,C 180,E1 -10928.756,E2 -10928.756} C_VEL
LIN {X 0,Y 404.139,Z 376.147,A -85,B 0,C 180,E1 -10931.602,E2 -10931.602} C_VEL
LIN {X 0,Y 404.153,Z 376.138,A -85,B 0,C 180,E1 -10934.523,E2 -10934.523} C_VEL
LIN {X 0,Y 404.203,Z 376.136,A -85,B 0,C 180,E1 -10937.304,E2 -10937.304} C_VEL
LIN {X 0,Y 404.164,Z 376.139,A -85,B 0,C 180,E1 -10939.955,E2 -10939.955} C_VEL
LIN {X 0,Y 404.135,Z 376.144,A -85,B 0,C 180,E1 -10943.124,E2 -10943.124} C_VEL
LIN {X 0,Y 404.139,Z 376.14,A -85,B 0,C 180,E1 -10946.187,E2 -10946.187} C_VEL
LIN {X 0,Y 404.147,Z 376.142,A -85,B 0,C 180,E1 -10949.715,E2 -10949.715} C_VEL
LIN {X 0,Y 404.189,Z 376.138,A -85,B 0,C 180,E1 -10953.122,E2 -10953.122} C_VEL
LIN {X 0,Y 404.171,Z 376.142,A -85,B 0,C 180,E1 -10955.334,E2 -10955.334} C_VEL
LIN {X 0,Y 404.133,Z 376.141,A -85,B 0,C 180,E1 -10958.58,E2 -10958.58} C_VEL
LIN {X 0,Y 404.203,Z 376.133,A -85,B 0,C 180,E1 -10961.762,E2 -10961.762} C_VEL
LIN {X 0,Y 404.199,Z 376.136,A -85,B 0,C 180,E1 -10964.882,E2 -10964.882} C_VEL
LIN {X 0,Y 404.263,Z 376.124,A -85,B 0,C 180,E1 -10967.959,E2 -10967.959} C_VEL
LIN {X 0,Y 404.425,Z 376.104,A -85,B 0,C 180,E1 -10972.1,E2 -10972.1} C_VEL
LIN {X 0,Y 404.416,Z 376.105,A -85,B 0,C 180,E1 -10974.015,E2 -10974.015} C_VEL
LIN {X 0,Y 404.475,Z 376.098,A -85,B 0,C 180,E1 -10978.009,E2 -10978.009} C_VEL
LIN {X 0,Y 404.605,Z 376.082,A -85,B 0,C 180,E1 -10980,E2 -10980} C_VEL
LIN {X 0,Y 404.417,Z 376.111,A -85,B 0,C 180,E1 -10982.988,E2 -10982.988} C_VEL
LIN {X 0,Y 404.404,Z 376.112,A -85,B 0,C 180,E1 -10986.987,E2 -10986.987} C_VEL
LIN {X 0,Y 404.263,Z 376.124,A -85,B 0,C 180,E1 -10990.012,E2 -10990.012} C_VEL
LIN {X 0,Y 404.258,Z 376.127,A -85,B 0,C 180,E1 -10993.212,E2 -10993.212} C_VEL
LIN {X 0,Y 404.208,Z 376.135,A -85,B 0,C 180,E1 -10997.007,E2 -10997.007} C_VEL
LIN {X 0,Y 404.18,Z 376.138,A -85,B 0,C 180,E1 -11000.351,E2 -11000.351} C_VEL
LIN {X 0,Y 404.163,Z 376.137,A -85,B 0,C 180,E1 -11003.575,E2 -11003.575} C_VEL
LIN {X 0,Y 404.177,Z 376.135,A -85,B 0,C 180,E1 -11005.767,E2 -11005.767} C_VEL
LIN {X 0,Y 404.189,Z 376.135,A -85,B 0,C 180,E1 -11008,E2 -11008} C_VEL
LIN {X 0,Y 404.133,Z 376.14,A -85,B 0,C 180,E1 -11011.559,E2 -11011.559} C_VEL
LIN {X 0,Y 404.18,Z 376.136,A -85,B 0,C 180,E1 -11015.017,E2 -11015.017} C_VEL
LIN {X 0,Y 404.158,Z 376.14,A -85,B 0,C 180,E1 -11018.757,E2 -11018.757} C_VEL
LIN {X 0,Y 404.187,Z 376.134,A -85,B 0,C 180,E1 -11021.611,E2 -11021.611} C_VEL
LIN {X 0,Y 404.186,Z 376.139,A -85,B 0,C 180,E1 -11024.529,E2 -11024.529} C_VEL
LIN {X 0,Y 404.135,Z 376.14,A -85,B 0,C 180,E1 -11027.297,E2 -11027.297} C_VEL
LIN {X 0,Y 404.167,Z 376.14,A -85,B 0,C 180,E1 -11029.956,E2 -11029.956} C_VEL
LIN {X 0,Y 404.138,Z 376.14,A -85,B 0,C 180,E1 -11033.125,E2 -11033.125} C_VEL
LIN {X 0,Y 404.144,Z 376.146,A -85,B 0,C 180,E1 -11036.189,E2 -11036.189} C_VEL
LIN {X 0,Y 404.145,Z 376.141,A -85,B 0,C 180,E1 -11039.716,E2 -11039.716} C_VEL
LIN {X 0,Y 404.195,Z 376.133,A -85,B 0,C 180,E1 -11043.124,E2 -11043.124} C_VEL
LIN {X 0,Y 404.177,Z 376.141,A -85,B 0,C 180,E1 -11045.335,E2 -11045.335} C_VEL
LIN {X 0,Y 404.188,Z 376.211,A -85,B 0,C 180,E1 -11046.784,E2 -11046.784} C_VEL
LIN {X 0,Y 406.071,Z 385.798,A -85,B 0,C 180,E1 -11049.378,E2 -11049.378} C_VEL
LIN {X 0,Y 406.314,Z 389.54,A -85,B 0,C 180,E1 -11050.331,E2 -11050.331} C_VEL
LIN {X 0,Y 410.698,Z 410.973,A -85,B 0,C 180,E1 -11050.962,E2 -11050.962} C_VEL
LIN {X 0,Y 409.562,Z 496.876,A -85,B 0,C 180,E1 -11052.493,E2 -11052.493} C_VEL
LIN {X 0,Y 409.045,Z 510.693,A -85,B 0,C 180,E1 -11052.953,E2 -11052.953} C_VEL
LIN {X 0,Y 408.473,Z 523.065,A -85,B 0,C 180,E1 -11053.572,E2 -11053.572} C_VEL
LIN {X 0,Y 407.803,Z 534.896,A -85,B 0,C 180,E1 -11054.379,E2 -11054.379} C_VEL
LIN {X 0,Y 407.037,Z 546.594,A -85,B 0,C 180,E1 -11055.409,E2 -11055.409} C_VEL
LIN {X 0,Y 406.315,Z 556.463,A -85,B 0,C 180,E1 -11056.497,E2 -11056.497} C_VEL
LIN {X 0,Y 405.492,Z 565.636,A -85,B 0,C 180,E1 -11057.742,E2 -11057.742} C_VEL
LIN {X 0,Y 404.739,Z 574.537,A -85,B 0,C 180,E1 -11059.242,E2 -11059.242} C_VEL
LIN {X 0,Y 404.128,Z 581.702,A -85,B 0,C 180,E1 -11060.743,E2 -11060.743} C_VEL
LIN {X 0,Y 403.721,Z 586.533,A -85,B 0,C 180,E1 -11061.995,E2 -11061.995} C_VEL
LIN {X 0,Y 403.464,Z 591.19,A -85,B 0,C 180,E1 -11063.487,E2 -11063.487} C_VEL
LIN {X 0,Y 403.138,Z 594.818,A -85,B 0,C 180,E1 -11065,E2 -11065} C_VEL
LIN {X 0,Y 403.036,Z 596.673,A -85,B 0,C 180,E1 -11066,E2 -11066} C_VEL
LIN {X 0,Y 403.015,Z 598.345,A -85,B 0,C 180,E1 -11067.28,E2 -11067.28} C_VEL
LIN {X 0,Y 402.887,Z 599.676,A -85,B 0,C 180,E1 -11069,E2 -11069} C_VEL
LIN {X 0,Y 402.873,Z 599.909,A -85,B 0,C 180,E1 -11070,E2 -11070} C_VEL
LIN {X 0,Y 402.922,Z 599.355,A -85,B 0,C 180,E1 -11071.625,E2 -11071.625} C_VEL
LIN {X 0,Y 402.325,Z 598.798,A -85,B 0,C 180,E1 -11072.456,E2 -11072.456} C_VEL
LIN {X 0,Y 399.552,Z 597.308,A -85,B 0,C 180,E1 -11073.799,E2 -11073.799} C_VEL
LIN {X 0,Y 397.227,Z 595.65,A -85,B 0,C 180,E1 -11074.87,E2 -11074.87} C_VEL
LIN {X 0,Y 396.301,Z 594.044,A -85,B 0,C 180,E1 -11075.683,E2 -11075.683} C_VEL
LIN {X 0,Y 396.266,Z 593.394,A -85,B 0,C 180,E1 -11075.955,E2 -11075.955} C_VEL
LIN {X 0,Y 396.565,Z 588.798,A -85,B 0,C 180,E1 -11077.638,E2 -11077.638} C_VEL
LIN {X 0,Y 397.07,Z 582.377,A -85,B 0,C 180,E1 -11079.423,E2 -11079.423} C_VEL
LIN {X 0,Y 397.701,Z 575.318,A -85,B 0,C 180,E1 -11080.951,E2 -11080.951} C_VEL
LIN {X 0,Y 398.496,Z 566.518,A -85,B 0,C 180,E1 -11082.477,E2 -11082.477} C_VEL
LIN {X 0,Y 399.344,Z 557.483,A -85,B 0,C 180,E1 -11083.744,E2 -11083.744} C_VEL
LIN {X 0,Y 400.107,Z 547.538,A -85,B 0,C 180,E1 -11084.88,E2 -11084.88} C_VEL
LIN {X 0,Y 400.91,Z 536.351,A -85,B 0,C 180,E1 -11085.897,E2 -11085.897} C_VEL
LIN {X 0,Y 401.702,Z 523.853,A -85,B 0,C 180,E1 -11086.778,E2 -11086.778} C_VEL
LIN {X 0,Y 402.334,Z 510.981,A -85,B 0,C 180,E1 -11087.438,E2 -11087.438} C_VEL
LIN {X 0,Y 402.865,Z 497.158,A -85,B 0,C 180,E1 -11087.906,E2 -11087.906} C_VEL
LIN {X 0,Y 403.291,Z 464.685,A -85,B 0,C 180,E1 -11088.514,E2 -11088.514} C_VEL
LIN {X 0,Y 403.958,Z 411.336,A -85,B 0,C 180,E1 -11089.465,E2 -11089.465} C_VEL
LIN {X 0,Y 399.395,Z 389.865,A -85,B 0,C 180,E1 -11090.112,E2 -11090.112} C_VEL
LIN {X 0,Y 398.027,Z 381.685,A -85,B 0,C 180,E1 -11092.31,E2 -11092.31} C_VEL
LIN {X 0,Y 397.146,Z 377.022,A -85,B 0,C 180,E1 -11093.634,E2 -11093.634} C_VEL
LIN {X 0,Y 397.195,Z 377.006,A -85,B 0,C 180,E1 -11097.389,E2 -11097.389} C_VEL
LIN {X 0,Y 397.078,Z 377.019,A -85,B 0,C 180,E1 -11100.882,E2 -11100.882} C_VEL
LIN {X 0,Y 397.125,Z 377.015,A -85,B 0,C 180,E1 -11104.492,E2 -11104.492} C_VEL
LIN {X 0,Y 397.105,Z 377.018,A -85,B 0,C 180,E1 -11108.274,E2 -11108.274} C_VEL
LIN {X 0,Y 397.087,Z 377.018,A -85,B 0,C 180,E1 -11110.908,E2 -11110.908} C_VEL
LIN {X 0,Y 397.1,Z 377.022,A -85,B 0,C 180,E1 -11113.647,E2 -11113.647} C_VEL
LIN {X 0,Y 397.156,Z 377.01,A -85,B 0,C 180,E1 -11116.511,E2 -11116.511} C_VEL
LIN {X 0,Y 397.119,Z 377.02,A -85,B 0,C 180,E1 -11119.55,E2 -11119.55} C_VEL
LIN {X 0,Y 397.094,Z 377.017,A -85,B 0,C 180,E1 -11122.789,E2 -11122.789} C_VEL
LIN {X 0,Y 397.113,Z 377.016,A -85,B 0,C 180,E1 -11126.281,E2 -11126.281} C_VEL
LIN {X 0,Y 397.099,Z 377.018,A -85,B 0,C 180,E1 -11130.135,E2 -11130.135} C_VEL
LIN {X 0,Y 397.188,Z 377.006,A -85,B 0,C 180,E1 -11132.609,E2 -11132.609} C_VEL
LIN {X 0,Y 397.127,Z 377.015,A -85,B 0,C 180,E1 -11135.981,E2 -11135.981} C_VEL
LIN {X 0,Y 397.137,Z 377.015,A -85,B 0,C 180,E1 -11139.702,E2 -11139.702} C_VEL
LIN {X 0,Y 397.174,Z 377.009,A -85,B 0,C 180,E1 -11142.844,E2 -11142.844} C_VEL
LIN {X 0,Y 397.219,Z 377.003,A -85,B 0,C 180,E1 -11146.679,E2 -11146.679} C_VEL
LIN {X 0,Y 397.221,Z 377.003,A -85,B 0,C 180,E1 -11149.809,E2 -11149.809} C_VEL
LIN {X 0,Y 397.355,Z 376.988,A -85,B 0,C 180,E1 -11152.888,E2 -11152.888} C_VEL
LIN {X 0,Y 397.249,Z 377.002,A -85,B 0,C 180,E1 -11154.925,E2 -11154.925} C_VEL
LIN {X 0,Y 397.444,Z 376.974,A -85,B 0,C 180,E1 -11157.973,E2 -11157.973} C_VEL
LIN {X 0,Y 397.574,Z 376.958,A -85,B 0,C 180,E1 -11160,E2 -11160} C_VEL
LIN {X 0,Y 397.376,Z 376.989,A -85,B 0,C 180,E1 -11163.041,E2 -11163.041} C_VEL
LIN {X 0,Y 397.356,Z 376.99,A -85,B 0,C 180,E1 -11167.112,E2 -11167.112} C_VEL
LIN {X 0,Y 397.222,Z 377.002,A -85,B 0,C 180,E1 -11170.191,E2 -11170.191} C_VEL
LIN {X 0,Y 397.219,Z 377.004,A -85,B 0,C 180,E1 -11173.321,E2 -11173.321} C_VEL
LIN {X 0,Y 397.174,Z 377.011,A -85,B 0,C 180,E1 -11177.155,E2 -11177.155} C_VEL
LIN {X 0,Y 397.096,Z 377.023,A -85,B 0,C 180,E1 -11180.73,E2 -11180.73} C_VEL
LIN {X 0,Y 397.126,Z 377.014,A -85,B 0,C 180,E1 -11184.019,E2 -11184.019} C_VEL
LIN {X 0,Y 397.188,Z 377.006,A -85,B 0,C 180,E1 -11187.391,E2 -11187.391} C_VEL
LIN {X 0,Y 397.072,Z 377.024,A -85,B 0,C 180,E1 -11190.883,E2 -11190.883} C_VEL
LIN {X 0,Y 397.12,Z 377.02,A -85,B 0,C 180,E1 -11194.494,E2 -11194.494} C_VEL
LIN {X 0,Y 397.105,Z 377.02,A -85,B 0,C 180,E1 -11198.275,E2 -11198.275} C_VEL
LIN {X 0,Y 397.151,Z 377.012,A -85,B 0,C 180,E1 -11201.994,E2 -11201.994} C_VEL
LIN {X 0,Y 397.109,Z 377.016,A -85,B 0,C 180,E1 -11205.066,E2 -11205.066} C_VEL
LIN {X 0,Y 397.076,Z 377.022,A -85,B 0,C 180,E1 -11208.02,E2 -11208.02} C_VEL
LIN {X 0,Y 397.131,Z 377.013,A -85,B 0,C 180,E1 -11211.139,E2 -11211.139} C_VEL
LIN {X 0,Y 397.118,Z 377.019,A -85,B 0,C 180,E1 -11214.497,E2 -11214.497} C_VEL
LIN {X 0,Y 397.079,Z 377.022,A -85,B 0,C 180,E1 -11217.929,E2 -11217.929} C_VEL
LIN {X 0,Y 397.161,Z 377.077,A -85,B 0,C 180,E1 -11221.171,E2 -11221.171} C_VEL
LIN {X 0,Y 399.645,Z 388.844,A -85,B 0,C 180,E1 -11223.92,E2 -11223.92} C_VEL
LIN {X 0,Y 400.682,Z 395.124,A -85,B 0,C 180,E1 -11225.332,E2 -11225.332} C_VEL
LIN {X 0,Y 399.372,Z 411.277,A -85,B 0,C 180,E1 -11228.685,E2 -11228.685} C_VEL
LIN {X 0,Y 398.969,Z 417.01,A -85,B 0,C 180,E1 -11229.877,E2 -11229.877} C_VEL
LIN {X 0,Y 403.499,Z 445.776,A -85,B 0,C 180,E1 -11230.663,E2 -11230.663} C_VEL
LIN {X 0,Y 402.534,Z 525.573,A -85,B 0,C 180,E1 -11232.111,E2 -11232.111} C_VEL
LIN {X 0,Y 401.974,Z 538.808,A -85,B 0,C 180,E1 -11232.546,E2 -11232.546} C_VEL
LIN {X 0,Y 401.293,Z 550.955,A -85,B 0,C 180,E1 -11233.139,E2 -11233.139} C_VEL
LIN {X 0,Y 400.368,Z 563.214,A -85,B 0,C 180,E1 -11233.951,E2 -11233.951} C_VEL
LIN {X 0,Y 399.432,Z 574.812,A -85,B 0,C 180,E1 -11234.958,E2 -11234.958} C_VEL
LIN {X 0,Y 398.595,Z 585.683,A -85,B 0,C 180,E1 -11236.151,E2 -11236.151} C_VEL
LIN {X 0,Y 397.825,Z 595.492,A -85,B 0,C 180,E1 -11237.502,E2 -11237.502} C_VEL
LIN {X 0,Y 396.991,Z 604.441,A -85,B 0,C 180,E1 -11239.029,E2 -11239.029} C_VEL
LIN {X 0,Y 396.476,Z 611.65,A -85,B 0,C 180,E1 -11240.563,E2 -11240.563} C_VEL
LIN {X 0,Y 396.173,Z 616.518,A -85,B 0,C 180,E1 -11241.841,E2 -11241.841} C_VEL
LIN {X 0,Y 395.919,Z 621.253,A -85,B 0,C 180,E1 -11243.375,E2 -11243.375} C_VEL
LIN {X 0,Y 395.842,Z 624.872,A -85,B 0,C 180,E1 -11244.907,E2 -11244.907} C_VEL
LIN {X 0,Y 395.777,Z 626.738,A -85,B 0,C 180,E1 -11245.927,E2 -11245.927} C_VEL
LIN {X 0,Y 395.804,Z 629.139,A -85,B 0,C 180,E1 -11247.965,E2 -11247.965} C_VEL
LIN {X 0,Y 395.81,Z 629.75,A -85,B 0,C 180,E1 -11248.983,E2 -11248.983} C_VEL
LIN {X 0,Y 395.798,Z 629.965,A -85,B 0,C 180,E1 -11250,E2 -11250} C_VEL
LIN {X 0,Y 395.81,Z 629.747,A -85,B 0,C 180,E1 -11251.017,E2 -11251.017} C_VEL
LIN {X 0,Y 395.804,Z 629.136,A -85,B 0,C 180,E1 -11252.035,E2 -11252.035} C_VEL
LIN {X 0,Y 395.777,Z 626.731,A -85,B 0,C 180,E1 -11254.073,E2 -11254.073} C_VEL
LIN {X 0,Y 395.826,Z 623.311,A -85,B 0,C 180,E1 -11255.805,E2 -11255.805} C_VEL
LIN {X 0,Y 396.064,Z 618.195,A -85,B 0,C 180,E1 -11257.648,E2 -11257.648} C_VEL
LIN {X 0,Y 396.405,Z 612.65,A -85,B 0,C 180,E1 -11259.181,E2 -11259.181} C_VEL
LIN {X 0,Y 396.863,Z 605.73,A -85,B 0,C 180,E1 -11260.716,E2 -11260.716} C_VEL
LIN {X 0,Y 397.668,Z 597.082,A -85,B 0,C 180,E1 -11262.244,E2 -11262.244} C_VEL
LIN {X 0,Y 398.358,Z 588.437,A -85,B 0,C 180,E1 -11263.489,E2 -11263.489} C_VEL
LIN {X 0,Y 399.201,Z 577.774,A -85,B 0,C 180,E1 -11264.737,E2 -11264.737} C_VEL
LIN {X 0,Y 400.14,Z 566.294,A -85,B 0,C 180,E1 -11265.797,E2 -11265.797} C_VEL
LIN {X 0,Y 401.049,Z 553.96,A -85,B 0,C 180,E1 -11266.675,E2 -11266.675} C_VEL
LIN {X 0,Y 401.762,Z 542.285,A -85,B 0,C 180,E1 -11267.3,E2 -11267.3} C_VEL
LIN {X 0,Y 402.382,Z 529.852,A -85,B 0,C 180,E1 -11267.764,E2 -11267.764} C_VEL
LIN {X 0,Y 402.764,Z 513.995,A -85,B 0,C 180,E1 -11268.108,E2 -11268.108} C_VEL
LIN {X 0,Y 403.425,Z 445.318,A -85,B 0,C 180,E1 -11269.34,E2 -11269.34} C_VEL
LIN {X 0,Y 398.934,Z 417.142,A -85,B 0,C 180,E1 -11270.091,E2 -11270.091} C_VEL
LIN {X 0,Y 400.245,Z 400.455,A -85,B 0,C 180,E1 -11273.545,E2 -11273.545} C_VEL
LIN {X 0,Y 400.586,Z 394.007,A -85,B 0,C 180,E1 -11274.901,E2 -11274.901} C_VEL
LIN {X 0,Y 398.353,Z 382.458,A -85,B 0,C 180,E1 -11277.543,E2 -11277.543} C_VEL
LIN {X 0,Y 397.152,Z 377.016,A -85,B 0,C 180,E1 -11278.866,E2 -11278.866} C_VEL
LIN {X 0,Y 397.078,Z 377.027,A -85,B 0,C 180,E1 -11282.071,E2 -11282.071} C_VEL
LIN {X 0,Y 397.118,Z 377.019,A -85,B 0,C 180,E1 -11285.503,E2 -11285.503} C_VEL
LIN {X 0,Y 397.131,Z 377.013,A -85,B 0,C 180,E1 -11288.861,E2 -11288.861} C_VEL
LIN {X 0,Y 397.075,Z 377.02,A -85,B 0,C 180,E1 -11292.265,E2 -11292.265} C_VEL
LIN {X 0,Y 397.114,Z 377.017,A -85,B 0,C 180,E1 -11295.064,E2 -11295.064} C_VEL
LIN {X 0,Y 397.151,Z 377.012,A -85,B 0,C 180,E1 -11298.006,E2 -11298.006} C_VEL
LIN {X 0,Y 397.105,Z 377.02,A -85,B 0,C 180,E1 -11301.725,E2 -11301.725} C_VEL
LIN {X 0,Y 397.12,Z 377.02,A -85,B 0,C 180,E1 -11305.506,E2 -11305.506} C_VEL
LIN {X 0,Y 397.079,Z 377.023,A -85,B 0,C 180,E1 -11309.117,E2 -11309.117} C_VEL
LIN {X 0,Y 397.188,Z 377.006,A -85,B 0,C 180,E1 -11312.609,E2 -11312.609} C_VEL
LIN {X 0,Y 397.126,Z 377.014,A -85,B 0,C 180,E1 -11315.981,E2 -11315.981} C_VEL
LIN {X 0,Y 397.131,Z 377.015,A -85,B 0,C 180,E1 -11319.704,E2 -11319.704} C_VEL
LIN {X 0,Y 397.174,Z 377.011,A -85,B 0,C 180,E1 -11322.845,E2 -11322.845} C_VEL
LIN {X 0,Y 397.221,Z 377.004,A -85,B 0,C 180,E1 -11326.702,E2 -11326.702} C_VEL
LIN {X 0,Y 397.222,Z 377.002,A -85,B 0,C 180,E1 -11329.809,E2 -11329.809} C_VEL
LIN {X 0,Y 397.355,Z 376.99,A -85,B 0,C 180,E1 -11332.888,E2 -11332.888} C_VEL
LIN {X 0,Y 397.249,Z 377.004,A -85,B 0,C 180,E1 -11334.925,E2 -11334.925} C_VEL
LIN {X 0,Y 397.444,Z 376.974,A -85,B 0,C 180,E1 -11337.973,E2 -11337.973} C_VEL
LIN {X 0,Y 397.574,Z 376.957,A -85,B 0,C 180,E1 -11340,E2 -11340} C_VEL
LIN {X 0,Y 397.375,Z 376.988,A -85,B 0,C 180,E1 -11343.041,E2 -11343.041} C_VEL
LIN {X 0,Y 397.356,Z 376.989,A -85,B 0,C 180,E1 -11347.112,E2 -11347.112} C_VEL
LIN {X 0,Y 397.221,Z 377.003,A -85,B 0,C 180,E1 -11350.191,E2 -11350.191} C_VEL
LIN {X 0,Y 397.219,Z 377.003,A -85,B 0,C 180,E1 -11353.321,E2 -11353.321} C_VEL
LIN {X 0,Y 397.174,Z 377.009,A -85,B 0,C 180,E1 -11357.156,E2 -11357.156} C_VEL
LIN {X 0,Y 397.107,Z 377.022,A -85,B 0,C 180,E1 -11360.73,E2 -11360.73} C_VEL
LIN {X 0,Y 397.127,Z 377.014,A -85,B 0,C 180,E1 -11364.019,E2 -11364.019} C_VEL
LIN {X 0,Y 397.188,Z 377.006,A -85,B 0,C 180,E1 -11367.391,E2 -11367.391} C_VEL
LIN {X 0,Y 397.072,Z 377.023,A -85,B 0,C 180,E1 -11370.883,E2 -11370.883} C_VEL
LIN {X 0,Y 397.12,Z 377.021,A -85,B 0,C 180,E1 -11374.494,E2 -11374.494} C_VEL
LIN {X 0,Y 397.105,Z 377.021,A -85,B 0,C 180,E1 -11378.275,E2 -11378.275} C_VEL
LIN {X 0,Y 397.152,Z 377.013,A -85,B 0,C 180,E1 -11381.994,E2 -11381.994} C_VEL
LIN {X 0,Y 397.107,Z 377.016,A -85,B 0,C 180,E1 -11385.066,E2 -11385.066} C_VEL
LIN {X 0,Y 397.065,Z 377.025,A -85,B 0,C 180,E1 -11388.022,E2 -11388.022} C_VEL
LIN {X 0,Y 397.132,Z 377.013,A -85,B 0,C 180,E1 -11391.139,E2 -11391.139} C_VEL
LIN {X 0,Y 397.119,Z 377.018,A -85,B 0,C 180,E1 -11394.497,E2 -11394.497} C_VEL
LIN {X 0,Y 397.078,Z 377.024,A -85,B 0,C 180,E1 -11397.929,E2 -11397.929} C_VEL
LIN {X 0,Y 397.122,Z 377.015,A -85,B 0,C 180,E1 -11401.457,E2 -11401.457} C_VEL
LIN {X 0,Y 397.153,Z 377.015,A -85,B 0,C 180,E1 -11404.488,E2 -11404.488} C_VEL
LIN {X 0,Y 397.151,Z 377.06,A -85,B 0,C 180,E1 -11406.509,E2 -11406.509} C_VEL
LIN {X 0,Y 399.181,Z 387.534,A -85,B 0,C 180,E1 -11409.383,E2 -11409.383} C_VEL
LIN {X 0,Y 399.407,Z 389.846,A -85,B 0,C 180,E1 -11409.987,E2 -11409.987} C_VEL
LIN {X 0,Y 403.993,Z 411.612,A -85,B 0,C 180,E1 -11410.64,E2 -11410.64} C_VEL
LIN {X 0,Y 402.826,Z 497.159,A -85,B 0,C 180,E1 -11412.19,E2 -11412.19} C_VEL
LIN {X 0,Y 402.276,Z 510.971,A -85,B 0,C 180,E1 -11412.657,E2 -11412.657} C_VEL
LIN {X 0,Y 401.686,Z 523.339,A -85,B 0,C 180,E1 -11413.286,E2 -11413.286} C_VEL
LIN {X 0,Y 400.994,Z 535.167,A -85,B 0,C 180,E1 -11414.107,E2 -11414.107} C_VEL
LIN {X 0,Y 400.25,Z 545.899,A -85,B 0,C 180,E1 -11415.058,E2 -11415.058} C_VEL
LIN {X 0,Y 399.432,Z 556.733,A -85,B 0,C 180,E1 -11416.259,E2 -11416.259} C_VEL
LIN {X 0,Y 398.566,Z 565.906,A -85,B 0,C 180,E1 -11417.526,E2 -11417.526} C_VEL
LIN {X 0,Y 397.754,Z 574.807,A -85,B 0,C 180,E1 -11419.051,E2 -11419.051} C_VEL
LIN {X 0,Y 397.107,Z 581.971,A -85,B 0,C 180,E1 -11420.578,E2 -11420.578} C_VEL
LIN {X 0,Y 396.683,Z 586.802,A -85,B 0,C 180,E1 -11421.852,E2 -11421.852} C_VEL
LIN {X 0,Y 396.387,Z 590.893,A -85,B 0,C 180,E1 -11423.165,E2 -11423.165} C_VEL
LIN {X 0,Y 396.086,Z 595.085,A -85,B 0,C 180,E1 -11424.91,E2 -11424.91} C_VEL
LIN {X 0,Y 395.953,Z 596.941,A -85,B 0,C 180,E1 -11425.929,E2 -11425.929} C_VEL
LIN {X 0,Y 395.956,Z 598.335,A -85,B 0,C 180,E1 -11426.948,E2 -11426.948} C_VEL
LIN {X 0,Y 395.9,Z 599.328,A -85,B 0,C 180,E1 -11427.965,E2 -11427.965} C_VEL
LIN {X 0,Y 395.799,Z 600.176,A -85,B 0,C 180,E1 -11430,E2 -11430} C_VEL
LIN {X 0,Y 395.901,Z 599.402,A -85,B 0,C 180,E1 -11432.035,E2 -11432.035} C_VEL
LIN {X 0,Y 395.955,Z 598.438,A -85,B 0,C 180,E1 -11433.052,E2 -11433.052} C_VEL
LIN {X 0,Y 395.951,Z 597.089,A -85,B 0,C 180,E1 -11434.071,E2 -11434.071} C_VEL
LIN {X 0,Y 396.266,Z 593.394,A -85,B 0,C 180,E1 -11435.955,E2 -11435.955} C_VEL
LIN {X 0,Y 395.742,Z 591.448,A -85,B 0,C 180,E1 -11436.758,E2 -11436.758} C_VEL
LIN {X 0,Y 393.12,Z 587.867,A -85,B 0,C 180,E1 -11438.048,E2 -11438.048} C_VEL
LIN {X 0,Y 390.619,Z 583.666,A -85,B 0,C 180,E1 -11439.311,E2 -11439.311} C_VEL
LIN {X 0,Y 390.289,Z 580.664,A -85,B 0,C 180,E1 -11440.059,E2 -11440.059} C_VEL
LIN {X 0,Y 391.05,Z 572.884,A -85,B 0,C 180,E1 -11441.665,E2 -11441.665} C_VEL
LIN {X 0,Y 391.716,Z 565.145,A -85,B 0,C 180,E1 -11442.96,E2 -11442.96} C_VEL
LIN {X 0,Y 392.781,Z 554.613,A -85,B 0,C 180,E1 -11444.374,E2 -11444.374} C_VEL
LIN {X 0,Y 393.574,Z 543.885,A -85,B 0,C 180,E1 -11445.536,E2 -11445.536} C_VEL
LIN {X 0,Y 394.367,Z 533.421,A -85,B 0,C 180,E1 -11446.433,E2 -11446.433} C_VEL
LIN {X 0,Y 395.139,Z 520.814,A -85,B 0,C 180,E1 -11447.265,E2 -11447.265} C_VEL
LIN {X 0,Y 395.73,Z 508.192,A -85,B 0,C 180,E1 -11447.873,E2 -11447.873} C_VEL
LIN {X 0,Y 396.129,Z 496.224,A -85,B 0,C 180,E1 -11448.255,E2 -11448.255} C_VEL
LIN {X 0,Y 397.289,Z 412.744,A -85,B 0,C 180,E1 -11449.784,E2 -11449.784} C_VEL
LIN {X 0,Y 392.841,Z 391.756,A -85,B 0,C 180,E1 -11450.422,E2 -11450.422} C_VEL
LIN {X 0,Y 392.396,Z 390.063,A -85,B 0,C 180,E1 -11450.504,E2 -11450.504} C_VEL
LIN {X 0,Y 390.112,Z 377.895,A -85,B 0,C 180,E1 -11453.912,E2 -11453.912} C_VEL
LIN {X 0,Y 390.114,Z 377.887,A -85,B 0,C 180,E1 -11456.767,E2 -11456.767} C_VEL
LIN {X 0,Y 390.039,Z 377.899,A -85,B 0,C 180,E1 -11460.299,E2 -11460.299} C_VEL
LIN {X 0,Y 390.067,Z 377.898,A -85,B 0,C 180,E1 -11464.024,E2 -11464.024} C_VEL
LIN {X 0,Y 390.044,Z 377.899,A -85,B 0,C 180,E1 -11467.55,E2 -11467.55} C_VEL
LIN {X 0,Y 390.054,Z 377.894,A -85,B 0,C 180,E1 -11470.821,E2 -11470.821} C_VEL
LIN {X 0,Y 390.057,Z 377.899,A -85,B 0,C 180,E1 -11473.886,E2 -11473.886} C_VEL
LIN {X 0,Y 390.11,Z 377.887,A -85,B 0,C 180,E1 -11476.797,E2 -11476.797} C_VEL
LIN {X 0,Y 390.073,Z 377.897,A -85,B 0,C 180,E1 -11479.562,E2 -11479.562} C_VEL
LIN {X 0,Y 390.042,Z 377.896,A -85,B 0,C 180,E1 -11482.448,E2 -11482.448} C_VEL
LIN {X 0,Y 390.063,Z 377.895,A -85,B 0,C 180,E1 -11486.044,E2 -11486.044} C_VEL
LIN {X 0,Y 390.04,Z 377.899,A -85,B 0,C 180,E1 -11489.868,E2 -11489.868} C_VEL
LIN {X 0,Y 390.107,Z 377.892,A -85,B 0,C 180,E1 -11493.231,E2 -11493.231} C_VEL
LIN {X 0,Y 390.1,Z 377.889,A -85,B 0,C 180,E1 -11496.75,E2 -11496.75} C_VEL
LIN {X 0,Y 390.1,Z 377.89,A -85,B 0,C 180,E1 -11499.983,E2 -11499.983} C_VEL
LIN {X 0,Y 390.13,Z 377.891,A -85,B 0,C 180,E1 -11503.248,E2 -11503.248} C_VEL
LIN {X 0,Y 390.187,Z 377.878,A -85,B 0,C 180,E1 -11506.561,E2 -11506.561} C_VEL
LIN {X 0,Y 390.171,Z 377.883,A -85,B 0,C 180,E1 -11509.623,E2 -11509.623} C_VEL
LIN {X 0,Y 390.31,Z 377.865,A -85,B 0,C 180,E1 -11512.759,E2 -11512.759} C_VEL
LIN {X 0,Y 390.22,Z 377.877,A -85,B 0,C 180,E1 -11514.833,E2 -11514.833} C_VEL
LIN {X 0,Y 390.413,Z 377.85,A -85,B 0,C 180,E1 -11517.937,E2 -11517.937} C_VEL
LIN {X 0,Y 390.544,Z 377.833,A -85,B 0,C 180,E1 -11520,E2 -11520} C_VEL
LIN {X 0,Y 390.31,Z 377.869,A -85,B 0,C 180,E1 -11523.097,E2 -11523.097} C_VEL
LIN {X 0,Y 390.323,Z 377.861,A -85,B 0,C 180,E1 -11526.202,E2 -11526.202} C_VEL
LIN {X 0,Y 390.307,Z 377.863,A -85,B 0,C 180,E1 -11528.282,E2 -11528.282} C_VEL
LIN {X 0,Y 390.171,Z 377.882,A -85,B 0,C 180,E1 -11532.483,E2 -11532.483} C_VEL
LIN {X 0,Y 390.132,Z 377.885,A -85,B 0,C 180,E1 -11535.677,E2 -11535.677} C_VEL
LIN {X 0,Y 390.098,Z 377.895,A -85,B 0,C 180,E1 -11538.922,E2 -11538.922} C_VEL
LIN {X 0,Y 390.033,Z 377.898,A -85,B 0,C 180,E1 -11542.235,E2 -11542.235} C_VEL
LIN {X 0,Y 390.112,Z 377.887,A -85,B 0,C 180,E1 -11545.744,E2 -11545.744} C_VEL
LIN {X 0,Y 390.052,Z 377.897,A -85,B 0,C 180,E1 -11549.11,E2 -11549.11} C_VEL
LIN {X 0,Y 390.037,Z 377.902,A -85,B 0,C 180,E1 -11552.722,E2 -11552.722} C_VEL
LIN {X 0,Y 390.052,Z 377.895,A -85,B 0,C 180,E1 -11555.826,E2 -11555.826} C_VEL
LIN {X 0,Y 390.07,Z 377.893,A -85,B 0,C 180,E1 -11559.22,E2 -11559.22} C_VEL
LIN {X 0,Y 390.116,Z 377.892,A -85,B 0,C 180,E1 -11562.387,E2 -11562.387} C_VEL
LIN {X 0,Y 390.06,Z 377.894,A -85,B 0,C 180,E1 -11565.358,E2 -11565.358} C_VEL
LIN {X 0,Y 390.069,Z 377.893,A -85,B 0,C 180,E1 -11569.177,E2 -11569.177} C_VEL
LIN {X 0,Y 390.044,Z 377.901,A -85,B 0,C 180,E1 -11572.449,E2 -11572.449} C_VEL
LIN {X 0,Y 390.067,Z 377.896,A -85,B 0,C 180,E1 -11575.976,E2 -11575.976} C_VEL
LIN {X 0,Y 390.039,Z 377.899,A -85,B 0,C 180,E1 -11579.701,E2 -11579.701} C_VEL
LIN {X 0,Y 390.109,Z 377.974,A -85,B 0,C 180,E1 -11580.858,E2 -11580.858} C_VEL
LIN {X 0,Y 392.511,Z 389.182,A -85,B 0,C 180,E1 -11583.543,E2 -11583.543} C_VEL
LIN {X 0,Y 393.763,Z 396.616,A -85,B 0,C 180,E1 -11585.248,E2 -11585.248} C_VEL
LIN {X 0,Y 392.353,Z 412.758,A -85,B 0,C 180,E1 -11588.662,E2 -11588.662} C_VEL
LIN {X 0,Y 392.059,Z 416.829,A -85,B 0,C 180,E1 -11589.524,E2 -11589.524} C_VEL
LIN {X 0,Y 396.862,Z 447.065,A -85,B 0,C 180,E1 -11590.356,E2 -11590.356} C_VEL
LIN {X 0,Y 395.786,Z 525.319,A -85,B 0,C 180,E1 -11591.796,E2 -11591.796} C_VEL
LIN {X 0,Y 395.203,Z 538.549,A -85,B 0,C 180,E1 -11592.237,E2 -11592.237} C_VEL
LIN {X 0,Y 394.5,Z 550.694,A -85,B 0,C 180,E1 -11592.839,E2 -11592.839} C_VEL
LIN {X 0,Y 393.538,Z 562.95,A -85,B 0,C 180,E1 -11593.664,E2 -11593.664} C_VEL
LIN {X 0,Y 392.555,Z 574.548,A -85,B 0,C 180,E1 -11594.689,E2 -11594.689} C_VEL
LIN {X 0,Y 391.699,Z 584.915,A -85,B 0,C 180,E1 -11595.84,E2 -11595.84} C_VEL
LIN {X 0,Y 391.018,Z 593.547,A -85,B 0,C 180,E1 -11597.017,E2 -11597.017} C_VEL
LIN {X 0,Y 390.264,Z 601.432,A -85,B 0,C 180,E1 -11598.312,E2 -11598.312} C_VEL
LIN {X 0,Y 389.618,Z 609.14,A -85,B 0,C 180,E1 -11599.871,E2 -11599.871} C_VEL
LIN {X 0,Y 389.117,Z 616.251,A -85,B 0,C 180,E1 -11601.692,E2 -11601.692} C_VEL
LIN {X 0,Y 388.843,Z 620.984,A -85,B 0,C 180,E1 -11603.253,E2 -11603.253} C_VEL
LIN {X 0,Y 388.738,Z 624.604,A -85,B 0,C 180,E1 -11604.814,E2 -11604.814} C_VEL
LIN {X 0,Y 388.701,Z 626.471,A -85,B 0,C 180,E1 -11605.853,E2 -11605.853} C_VEL
LIN {X 0,Y 388.702,Z 628.872,A -85,B 0,C 180,E1 -11607.928,E2 -11607.928} C_VEL
LIN {X 0,Y 388.739,Z 629.484,A -85,B 0,C 180,E1 -11608.964,E2 -11608.964} C_VEL
LIN {X 0,Y 388.726,Z 629.699,A -85,B 0,C 180,E1 -11610,E2 -11610} C_VEL
LIN {X 0,Y 388.739,Z 629.481,A -85,B 0,C 180,E1 -11611.036,E2 -11611.036} C_VEL
LIN {X 0,Y 388.703,Z 628.869,A -85,B 0,C 180,E1 -11612.072,E2 -11612.072} C_VEL
LIN {X 0,Y 388.701,Z 626.464,A -85,B 0,C 180,E1 -11614.147,E2 -11614.147} C_VEL
LIN {X 0,Y 388.726,Z 623.414,A -85,B 0,C 180,E1 -11615.753,E2 -11615.753} C_VEL
LIN {X 0,Y 388.933,Z 619.526,A -85,B 0,C 180,E1 -11617.267,E2 -11617.267} C_VEL
LIN {X 0,Y 389.304,Z 613.396,A -85,B 0,C 180,E1 -11619.088,E2 -11619.088} C_VEL
LIN {X 0,Y 389.772,Z 606.7,A -85,B 0,C 180,E1 -11620.65,E2 -11620.65} C_VEL
LIN {X 0,Y 390.547,Z 598.402,A -85,B 0,C 180,E1 -11622.207,E2 -11622.207} C_VEL
LIN {X 0,Y 391.264,Z 589.895,A -85,B 0,C 180,E1 -11623.503,E2 -11623.503} C_VEL
LIN {X 0,Y 392.155,Z 579.387,A -85,B 0,C 180,E1 -11624.796,E2 -11624.796} C_VEL
LIN {X 0,Y 393.172,Z 567.568,A -85,B 0,C 180,E1 -11625.952,E2 -11625.952} C_VEL
LIN {X 0,Y 394.108,Z 555.68,A -85,B 0,C 180,E1 -11626.844,E2 -11626.844} C_VEL
LIN {X 0,Y 394.888,Z 543.313,A -85,B 0,C 180,E1 -11627.544,E2 -11627.544} C_VEL
LIN {X 0,Y 395.593,Z 530.613,A -85,B 0,C 180,E1 -11628.046,E2 -11628.046} C_VEL
LIN {X 0,Y 395.918,Z 517.287,A -85,B 0,C 180,E1 -11628.365,E2 -11628.365} C_VEL
LIN {X 0,Y 396.747,Z 446.321,A -85,B 0,C 180,E1 -11629.655,E2 -11629.655} C_VEL
LIN {X 0,Y 392.052,Z 416.873,A -85,B 0,C 180,E1 -11630.459,E2 -11630.459} C_VEL
LIN {X 0,Y 393.46,Z 400.203,A -85,B 0,C 180,E1 -11633.976,E2 -11633.976} C_VEL
LIN {X 0,Y 393.601,Z 395.032,A -85,B 0,C 180,E1 -11635.093,E2 -11635.093} C_VEL
LIN {X 0,Y 391.322,Z 383.314,A -85,B 0,C 180,E1 -11637.836,E2 -11637.836} C_VEL
LIN {X 0,Y 390.107,Z 377.894,A -85,B 0,C 180,E1 -11639.179,E2 -11639.179} C_VEL
LIN {X 0,Y 390.042,Z 377.9,A -85,B 0,C 180,E1 -11642.721,E2 -11642.721} C_VEL
LIN {X 0,Y 390.055,Z 377.899,A -85,B 0,C 180,E1 -11645.825,E2 -11645.825} C_VEL
LIN {X 0,Y 390.069,Z 377.895,A -85,B 0,C 180,E1 -11649.218,E2 -11649.218} C_VEL
LIN {X 0,Y 390.047,Z 377.895,A -85,B 0,C 180,E1 -11652.375,E2 -11652.375} C_VEL
LIN {X 0,Y 390.098,Z 377.89,A -85,B 0,C 180,E1 -11656.106,E2 -11656.106} C_VEL
LIN {X 0,Y 390.078,Z 377.895,A -85,B 0,C 180,E1 -11659.173,E2 -11659.173} C_VEL
LIN {X 0,Y 390.042,Z 377.896,A -85,B 0,C 180,E1 -11662.448,E2 -11662.448} C_VEL
LIN {X 0,Y 390.062,Z 377.894,A -85,B 0,C 180,E1 -11666.045,E2 -11666.045} C_VEL
LIN {X 0,Y 390.046,Z 377.897,A -85,B 0,C 180,E1 -11669.867,E2 -11669.867} C_VEL
LIN {X 0,Y 390.107,Z 377.894,A -85,B 0,C 180,E1 -11673.231,E2 -11673.231} C_VEL
LIN {X 0,Y 390.1,Z 377.89,A -85,B 0,C 180,E1 -11676.75,E2 -11676.75} C_VEL
LIN {X 0,Y 390.097,Z 377.889,A -85,B 0,C 180,E1 -11679.983,E2 -11679.983} C_VEL
LIN {X 0,Y 390.13,Z 377.891,A -85,B 0,C 180,E1 -11683.248,E2 -11683.248} C_VEL
LIN {X 0,Y 390.187,Z 377.879,A -85,B 0,C 180,E1 -11686.561,E2 -11686.561} C_VEL
LIN {X 0,Y 390.171,Z 377.881,A -85,B 0,C 180,E1 -11689.623,E2 -11689.623} C_VEL
LIN {X 0,Y 390.31,Z 377.866,A -85,B 0,C 180,E1 -11692.759,E2 -11692.759} C_VEL
LIN {X 0,Y 390.22,Z 377.878,A -85,B 0,C 180,E1 -11694.833,E2 -11694.833} C_VEL
LIN {X 0,Y 390.413,Z 377.85,A -85,B 0,C 180,E1 -11697.937,E2 -11697.937} C_VEL
LIN {X 0,Y 390.544,Z 377.833,A -85,B 0,C 180,E1 -11700,E2 -11700} C_VEL
LIN {X 0,Y 390.31,Z 377.867,A -85,B 0,C 180,E1 -11703.097,E2 -11703.097} C_VEL
LIN {X 0,Y 390.302,Z 377.863,A -85,B 0,C 180,E1 -11706.66,E2 -11706.66} C_VEL
LIN {X 0,Y 390.202,Z 377.878,A -85,B 0,C 180,E1 -11709.329,E2 -11709.329} C_VEL
LIN {X 0,Y 390.17,Z 377.883,A -85,B 0,C 180,E1 -11712.483,E2 -11712.483} C_VEL
LIN {X 0,Y 390.132,Z 377.885,A -85,B 0,C 180,E1 -11715.677,E2 -11715.677} C_VEL
LIN {X 0,Y 390.098,Z 377.893,A -85,B 0,C 180,E1 -11718.923,E2 -11718.923} C_VEL
LIN {X 0,Y 390.034,Z 377.899,A -85,B 0,C 180,E1 -11722.235,E2 -11722.235} C_VEL
LIN {X 0,Y 390.113,Z 377.887,A -85,B 0,C 180,E1 -11725.744,E2 -11725.744} C_VEL
LIN {X 0,Y 390.052,Z 377.896,A -85,B 0,C 180,E1 -11729.11,E2 -11729.11} C_VEL
LIN {X 0,Y 390.037,Z 377.901,A -85,B 0,C 180,E1 -11732.722,E2 -11732.722} C_VEL
LIN {X 0,Y 390.052,Z 377.895,A -85,B 0,C 180,E1 -11735.826,E2 -11735.826} C_VEL
LIN {X 0,Y 390.07,Z 377.893,A -85,B 0,C 180,E1 -11739.22,E2 -11739.22} C_VEL
LIN {X 0,Y 390.117,Z 377.893,A -85,B 0,C 180,E1 -11742.388,E2 -11742.388} C_VEL
LIN {X 0,Y 390.058,Z 377.894,A -85,B 0,C 180,E1 -11745.358,E2 -11745.358} C_VEL
LIN {X 0,Y 390.029,Z 377.903,A -85,B 0,C 180,E1 -11748.188,E2 -11748.188} C_VEL
LIN {X 0,Y 390.09,Z 377.891,A -85,B 0,C 180,E1 -11750.909,E2 -11750.909} C_VEL
LIN {X 0,Y 390.085,Z 377.892,A -85,B 0,C 180,E1 -11754.794,E2 -11754.794} C_VEL
LIN {X 0,Y 390.031,Z 377.901,A -85,B 0,C 180,E1 -11757.876,E2 -11757.876} C_VEL
LIN {X 0,Y 390.058,Z 377.894,A -85,B 0,C 180,E1 -11760.891,E2 -11760.891} C_VEL
LIN {X 0,Y 390.119,Z 377.892,A -85,B 0,C 180,E1 -11764.257,E2 -11764.257} C_VEL
LIN {X 0,Y 390.092,Z 377.994,A -85,B 0,C 180,E1 -11766.242,E2 -11766.242} C_VEL
LIN {X 0,Y 392.262,Z 389.103,A -85,B 0,C 180,E1 -11769.342,E2 -11769.342} C_VEL
LIN {X 0,Y 392.411,Z 390.327,A -85,B 0,C 180,E1 -11769.628,E2 -11769.628} C_VEL
LIN {X 0,Y 396.399,Z 407.864,A -85,B 0,C 180,E1 -11770.177,E2 -11770.177} C_VEL
LIN {X 0,Y 397.309,Z 412.987,A -85,B 0,C 180,E1 -11770.321,E2 -11770.321} C_VEL
LIN {X 0,Y 396.081,Z 497.442,A -85,B 0,C 180,E1 -11771.877,E2 -11771.877} C_VEL
LIN {X 0,Y 395.517,Z 511.249,A -85,B 0,C 180,E1 -11772.351,E2 -11772.351} C_VEL
LIN {X 0,Y 394.912,Z 523.613,A -85,B 0,C 180,E1 -11772.991,E2 -11772.991} C_VEL
LIN {X 0,Y 394.181,Z 535.44,A -85,B 0,C 180,E1 -11773.825,E2 -11773.825} C_VEL
LIN {X 0,Y 393.37,Z 546.697,A -85,B 0,C 180,E1 -11774.845,E2 -11774.845} C_VEL
LIN {X 0,Y 392.551,Z 557.003,A -85,B 0,C 180,E1 -11776.014,E2 -11776.014} C_VEL
LIN {X 0,Y 391.653,Z 566.175,A -85,B 0,C 180,E1 -11777.302,E2 -11777.302} C_VEL
LIN {X 0,Y 390.794,Z 575.077,A -85,B 0,C 180,E1 -11778.853,E2 -11778.853} C_VEL
LIN {X 0,Y 390.11,Z 582.24,A -85,B 0,C 180,E1 -11780.408,E2 -11780.408} C_VEL
LIN {X 0,Y 389.668,Z 587.07,A -85,B 0,C 180,E1 -11781.704,E2 -11781.704} C_VEL
LIN {X 0,Y 389.304,Z 591.516,A -85,B 0,C 180,E1 -11783.17,E2 -11783.17} C_VEL
LIN {X 0,Y 389.038,Z 595.352,A -85,B 0,C 180,E1 -11784.818,E2 -11784.818} C_VEL
LIN {X 0,Y 388.874,Z 597.209,A -85,B 0,C 180,E1 -11785.855,E2 -11785.855} C_VEL
LIN {X 0,Y 388.862,Z 598.603,A -85,B 0,C 180,E1 -11786.892,E2 -11786.892} C_VEL
LIN {X 0,Y 388.818,Z 599.595,A -85,B 0,C 180,E1 -11787.928,E2 -11787.928} C_VEL
LIN {X 0,Y 388.727,Z 600.442,A -85,B 0,C 180,E1 -11790,E2 -11790} C_VEL
LIN {X 0,Y 388.747,Z 600.253,A -85,B 0,C 180,E1 -11791.036,E2 -11791.036} C_VEL
LIN {X 0,Y 388.818,Z 599.669,A -85,B 0,C 180,E1 -11792.072,E2 -11792.072} C_VEL
LIN {X 0,Y 388.861,Z 598.705,A -85,B 0,C 180,E1 -11793.108,E2 -11793.108} C_VEL
LIN {X 0,Y 388.873,Z 597.355,A -85,B 0,C 180,E1 -11794.145,E2 -11794.145} C_VEL
LIN {X 0,Y 389.207,Z 593.805,A -85,B 0,C 180,E1 -11796,E2 -11796} C_VEL
LIN {X 0,Y 389.531,Z 589.064,A -85,B 0,C 180,E1 -11797.777,E2 -11797.777} C_VEL
LIN {X 0,Y 390.077,Z 582.642,A -85,B 0,C 180,E1 -11799.593,E2 -11799.593} C_VEL
LIN {X 0,Y 390.289,Z 580.664,A -85,B 0,C 180,E1 -11800.059,E2 -11800.059} C_VEL
LIN {X 0,Y 389.986,Z 577.478,A -85,B 0,C 180,E1 -11800.786,E2 -11800.786} C_VEL
LIN {X 0,Y 387.673,Z 571.992,A -85,B 0,C 180,E1 -11801.954,E2 -11801.954} C_VEL
LIN {X 0,Y 385.428,Z 566.02,A -85,B 0,C 180,E1 -11803.073,E2 -11803.073} C_VEL
LIN {X 0,Y 385.232,Z 561.909,A -85,B 0,C 180,E1 -11803.712,E2 -11803.712} C_VEL
LIN {X 0,Y 386.103,Z 552.285,A -85,B 0,C 180,E1 -11804.949,E2 -11804.949} C_VEL
LIN {X 0,Y 386.904,Z 541.346,A -85,B 0,C 180,E1 -11806.082,E2 -11806.082} C_VEL
LIN {X 0,Y 387.81,Z 530.164,A -85,B 0,C 180,E1 -11806.991,E2 -11806.991} C_VEL
LIN {X 0,Y 388.531,Z 518.816,A -85,B 0,C 180,E1 -11807.704,E2 -11807.704} C_VEL
LIN {X 0,Y 389.093,Z 505.861,A -85,B 0,C 180,E1 -11808.29,E2 -11808.29} C_VEL
LIN {X 0,Y 389.438,Z 493.493,A -85,B 0,C 180,E1 -11808.648,E2 -11808.648} C_VEL
LIN {X 0,Y 390.554,Z 413.093,A -85,B 0,C 180,E1 -11810.138,E2 -11810.138} C_VEL
LIN {X 0,Y 386.258,Z 393.315,A -85,B 0,C 180,E1 -11810.76,E2 -11810.76} C_VEL
LIN {X 0,Y 385.248,Z 390.316,A -85,B 0,C 180,E1 -11810.907,E2 -11810.907} C_VEL
LIN {X 0,Y 383.059,Z 378.773,A -85,B 0,C 180,E1 -11814.201,E2 -11814.201} C_VEL
LIN {X 0,Y 383.057,Z 378.767,A -85,B 0,C 180,E1 -11817.301,E2 -11817.301} C_VEL
LIN {X 0,Y 382.983,Z 378.775,A -85,B 0,C 180,E1 -11820.918,E2 -11820.918} C_VEL
LIN {X 0,Y 383.017,Z 378.771,A -85,B 0,C 180,E1 -11824.667,E2 -11824.667} C_VEL
LIN {X 0,Y 383,Z 378.779,A -85,B 0,C 180,E1 -11827.903,E2 -11827.903} C_VEL
LIN {X 0,Y 382.982,Z 378.777,A -85,B 0,C 180,E1 -11831.346,E2 -11831.346} C_VEL
LIN {X 0,Y 383.005,Z 378.774,A -85,B 0,C 180,E1 -11834.304,E2 -11834.304} C_VEL
LIN {X 0,Y 383.072,Z 378.766,A -85,B 0,C 180,E1 -11837.248,E2 -11837.248} C_VEL
LIN {X 0,Y 383.018,Z 378.771,A -85,B 0,C 180,E1 -11840.411,E2 -11840.411} C_VEL
LIN {X 0,Y 383.022,Z 378.773,A -85,B 0,C 180,E1 -11844.044,E2 -11844.044} C_VEL
LIN {X 0,Y 383,Z 378.78,A -85,B 0,C 180,E1 -11847.573,E2 -11847.573} C_VEL
LIN {X 0,Y 382.986,Z 378.775,A -85,B 0,C 180,E1 -11850.299,E2 -11850.299} C_VEL
LIN {X 0,Y 383.05,Z 378.767,A -85,B 0,C 180,E1 -11852.697,E2 -11852.697} C_VEL
LIN {X 0,Y 383.027,Z 378.77,A -85,B 0,C 180,E1 -11856.192,E2 -11856.192} C_VEL
LIN {X 0,Y 383.053,Z 378.771,A -85,B 0,C 180,E1 -11859.598,E2 -11859.598} C_VEL
LIN {X 0,Y 383.097,Z 378.763,A -85,B 0,C 180,E1 -11862.931,E2 -11862.931} C_VEL
LIN {X 0,Y 383.118,Z 378.758,A -85,B 0,C 180,E1 -11866.463,E2 -11866.463} C_VEL
LIN {X 0,Y 383.133,Z 378.761,A -85,B 0,C 180,E1 -11869.43,E2 -11869.43} C_VEL
LIN {X 0,Y 383.265,Z 378.741,A -85,B 0,C 180,E1 -11872.625,E2 -11872.625} C_VEL
LIN {X 0,Y 383.192,Z 378.751,A -85,B 0,C 180,E1 -11874.738,E2 -11874.738} C_VEL
LIN {X 0,Y 383.38,Z 378.726,A -85,B 0,C 180,E1 -11877.899,E2 -11877.899} C_VEL
LIN {X 0,Y 383.513,Z 378.709,A -85,B 0,C 180,E1 -11880,E2 -11880} C_VEL
LIN {X 0,Y 383.246,Z 378.748,A -85,B 0,C 180,E1 -11883.154,E2 -11883.154} C_VEL
LIN {X 0,Y 383.28,Z 378.739,A -85,B 0,C 180,E1 -11886.316,E2 -11886.316} C_VEL
LIN {X 0,Y 383.253,Z 378.743,A -85,B 0,C 180,E1 -11888.436,E2 -11888.436} C_VEL
LIN {X 0,Y 383.1,Z 378.761,A -85,B 0,C 180,E1 -11891.642,E2 -11891.642} C_VEL
LIN {X 0,Y 383.104,Z 378.767,A -85,B 0,C 180,E1 -11894.882,E2 -11894.882} C_VEL
LIN {X 0,Y 383.055,Z 378.767,A -85,B 0,C 180,E1 -11898.174,E2 -11898.174} C_VEL
LIN {X 0,Y 382.986,Z 378.775,A -85,B 0,C 180,E1 -11901.531,E2 -11901.531} C_VEL
LIN {X 0,Y 383.046,Z 378.772,A -85,B 0,C 180,E1 -11904.961,E2 -11904.961} C_VEL
LIN {X 0,Y 383.034,Z 378.773,A -85,B 0,C 180,E1 -11908.493,E2 -11908.493} C_VEL
LIN {X 0,Y 383.003,Z 378.774,A -85,B 0,C 180,E1 -11912.15,E2 -11912.15} C_VEL
LIN {X 0,Y 383.013,Z 378.778,A -85,B 0,C 180,E1 -11914.669,E2 -11914.669} C_VEL
LIN {X 0,Y 382.998,Z 378.774,A -85,B 0,C 180,E1 -11917.905,E2 -11917.905} C_VEL
LIN {X 0,Y 383.042,Z 378.768,A -85,B 0,C 180,E1 -11921.34,E2 -11921.34} C_VEL
LIN {X 0,Y 383.031,Z 378.774,A -85,B 0,C 180,E1 -11924.31,E2 -11924.31} C_VEL
LIN {X 0,Y 383.007,Z 378.772,A -85,B 0,C 180,E1 -11927.241,E2 -11927.241} C_VEL
LIN {X 0,Y 383.016,Z 378.778,A -85,B 0,C 180,E1 -11930.414,E2 -11930.414} C_VEL
LIN {X 0,Y 383.025,Z 378.773,A -85,B 0,C 180,E1 -11934.045,E2 -11934.045} C_VEL
LIN {X 0,Y 382.987,Z 378.775,A -85,B 0,C 180,E1 -11937.578,E2 -11937.578} C_VEL
LIN {X 0,Y 383.062,Z 378.853,A -85,B 0,C 180,E1 -11940.534,E2 -11940.534} C_VEL
LIN {X 0,Y 385.504,Z 390.117,A -85,B 0,C 180,E1 -11943.292,E2 -11943.292} C_VEL
LIN {X 0,Y 386.797,Z 397.439,A -85,B 0,C 180,E1 -11945.012,E2 -11945.012} C_VEL
LIN {X 0,Y 385.621,Z 411.501,A -85,B 0,C 180,E1 -11948.051,E2 -11948.051} C_VEL
LIN {X 0,Y 385.18,Z 416.608,A -85,B 0,C 180,E1 -11949.149,E2 -11949.149} C_VEL
LIN {X 0,Y 390.101,Z 447.395,A -85,B 0,C 180,E1 -11950.012,E2 -11950.012} C_VEL
LIN {X 0,Y 389.051,Z 525.064,A -85,B 0,C 180,E1 -11951.469,E2 -11951.469} C_VEL
LIN {X 0,Y 388.462,Z 538.29,A -85,B 0,C 180,E1 -11951.918,E2 -11951.918} C_VEL
LIN {X 0,Y 387.694,Z 550.432,A -85,B 0,C 180,E1 -11952.528,E2 -11952.528} C_VEL
LIN {X 0,Y 386.717,Z 562.687,A -85,B 0,C 180,E1 -11953.368,E2 -11953.368} C_VEL
LIN {X 0,Y 385.697,Z 574.284,A -85,B 0,C 180,E1 -11954.409,E2 -11954.409} C_VEL
LIN {X 0,Y 384.831,Z 583.582,A -85,B 0,C 180,E1 -11955.448,E2 -11955.448} C_VEL
LIN {X 0,Y 384.065,Z 593.28,A -85,B 0,C 180,E1 -11956.778,E2 -11956.778} C_VEL
LIN {X 0,Y 383.302,Z 601.167,A -85,B 0,C 180,E1 -11958.096,E2 -11958.096} C_VEL
LIN {X 0,Y 382.598,Z 608.873,A -85,B 0,C 180,E1 -11959.683,E2 -11959.683} C_VEL
LIN {X 0,Y 382.052,Z 615.984,A -85,B 0,C 180,E1 -11961.538,E2 -11961.538} C_VEL
LIN {X 0,Y 381.78,Z 620.718,A -85,B 0,C 180,E1 -11963.128,E2 -11963.128} C_VEL
LIN {X 0,Y 381.639,Z 624.337,A -85,B 0,C 180,E1 -11964.717,E2 -11964.717} C_VEL
LIN {X 0,Y 381.626,Z 626.205,A -85,B 0,C 180,E1 -11965.776,E2 -11965.776} C_VEL
LIN {X 0,Y 381.601,Z 628.605,A -85,B 0,C 180,E1 -11967.889,E2 -11967.889} C_VEL
LIN {X 0,Y 381.67,Z 629.218,A -85,B 0,C 180,E1 -11968.945,E2 -11968.945} C_VEL
LIN {X 0,Y 381.657,Z 629.433,A -85,B 0,C 180,E1 -11970,E2 -11970} C_VEL
LIN {X 0,Y 381.67,Z 629.215,A -85,B 0,C 180,E1 -11971.055,E2 -11971.055} C_VEL
LIN {X 0,Y 381.601,Z 628.601,A -85,B 0,C 180,E1 -11972.111,E2 -11972.111} C_VEL
LIN {X 0,Y 381.626,Z 626.196,A -85,B 0,C 180,E1 -11974.224,E2 -11974.224} C_VEL
LIN {X 0,Y 381.687,Z 622.545,A -85,B 0,C 180,E1 -11976.118,E2 -11976.118} C_VEL
LIN {X 0,Y 381.941,Z 617.657,A -85,B 0,C 180,E1 -11977.932,E2 -11977.932} C_VEL
LIN {X 0,Y 382.326,Z 612.11,A -85,B 0,C 180,E1 -11979.523,E2 -11979.523} C_VEL
LIN {X 0,Y 382.864,Z 605.19,A -85,B 0,C 180,E1 -11981.113,E2 -11981.113} C_VEL
LIN {X 0,Y 383.765,Z 596.541,A -85,B 0,C 180,E1 -11982.695,E2 -11982.695} C_VEL
LIN {X 0,Y 384.639,Z 586.906,A -85,B 0,C 180,E1 -11984.115,E2 -11984.115} C_VEL
LIN {X 0,Y 385.477,Z 576.758,A -85,B 0,C 180,E1 -11985.329,E2 -11985.329} C_VEL
LIN {X 0,Y 386.473,Z 565.75,A -85,B 0,C 180,E1 -11986.371,E2 -11986.371} C_VEL
LIN {X 0,Y 387.453,Z 553.414,A -85,B 0,C 180,E1 -11987.279,E2 -11987.279} C_VEL
LIN {X 0,Y 388.221,Z 541.736,A -85,B 0,C 180,E1 -11987.923,E2 -11987.923} C_VEL
LIN {X 0,Y 388.89,Z 529.293,A -85,B 0,C 180,E1 -11988.402,E2 -11988.402} C_VEL
LIN {X 0,Y 389.319,Z 513.423,A -85,B 0,C 180,E1 -11988.756,E2 -11988.756} C_VEL
LIN {X 0,Y 390.063,Z 447.149,A -85,B 0,C 180,E1 -11989.985,E2 -11989.985} C_VEL
LIN {X 0,Y 385.152,Z 416.546,A -85,B 0,C 180,E1 -11990.855,E2 -11990.855} C_VEL
LIN {X 0,Y 386.544,Z 401.238,A -85,B 0,C 180,E1 -11994.147,E2 -11994.147} C_VEL
LIN {X 0,Y 386.786,Z 397.37,A -85,B 0,C 180,E1 -11994.989,E2 -11994.989} C_VEL
LIN {X 0,Y 384.585,Z 385.663,A -85,B 0,C 180,E1 -11997.774,E2 -11997.774} C_VEL
LIN {X 0,Y 383.042,Z 378.774,A -85,B 0,C 180,E1 -11999.506,E2 -11999.506} C_VEL
LIN {X 0,Y 383.002,Z 378.777,A -85,B 0,C 180,E1 -12003.4,E2 -12003.4} C_VEL
LIN {X 0,Y 383.032,Z 378.771,A -85,B 0,C 180,E1 -12006.164,E2 -12006.164} C_VEL
LIN {X 0,Y 383.013,Z 378.775,A -85,B 0,C 180,E1 -12009.957,E2 -12009.957} C_VEL
LIN {X 0,Y 383.002,Z 378.773,A -85,B 0,C 180,E1 -12012.778,E2 -12012.778} C_VEL
LIN {X 0,Y 383.035,Z 378.773,A -85,B 0,C 180,E1 -12015.795,E2 -12015.795} C_VEL
LIN {X 0,Y 383.04,Z 378.769,A -85,B 0,C 180,E1 -12018.786,E2 -12018.786} C_VEL
LIN {X 0,Y 382.998,Z 378.774,A -85,B 0,C 180,E1 -12022.095,E2 -12022.095} C_VEL
LIN {X 0,Y 383.013,Z 378.777,A -85,B 0,C 180,E1 -12025.331,E2 -12025.331} C_VEL
LIN {X 0,Y 382.98,Z 378.779,A -85,B 0,C 180,E1 -12029.081,E2 -12029.081} C_VEL
LIN {X 0,Y 383.05,Z 378.768,A -85,B 0,C 180,E1 -12032.698,E2 -12032.698} C_VEL
LIN {X 0,Y 383.027,Z 378.77,A -85,B 0,C 180,E1 -12036.192,E2 -12036.192} C_VEL
LIN {X 0,Y 383.048,Z 378.77,A -85,B 0,C 180,E1 -12039.598,E2 -12039.598} C_VEL
LIN {X 0,Y 383.097,Z 378.765,A -85,B 0,C 180,E1 -12042.931,E2 -12042.931} C_VEL
LIN {X 0,Y 383.118,Z 378.759,A -85,B 0,C 180,E1 -12046.463,E2 -12046.463} C_VEL
LIN {X 0,Y 383.133,Z 378.759,A -85,B 0,C 180,E1 -12049.43,E2 -12049.43} C_VEL
LIN {X 0,Y 383.265,Z 378.742,A -85,B 0,C 180,E1 -12052.625,E2 -12052.625} C_VEL
LIN {X 0,Y 383.192,Z 378.753,A -85,B 0,C 180,E1 -12054.738,E2 -12054.738} C_VEL
LIN {X 0,Y 383.38,Z 378.726,A -85,B 0,C 180,E1 -12057.899,E2 -12057.899} C_VEL
LIN {X 0,Y 383.513,Z 378.709,A -85,B 0,C 180,E1 -12060,E2 -12060} C_VEL
LIN {X 0,Y 383.246,Z 378.746,A -85,B 0,C 180,E1 -12063.154,E2 -12063.154} C_VEL
LIN {X 0,Y 383.261,Z 378.74,A -85,B 0,C 180,E1 -12066.654,E2 -12066.654} C_VEL
LIN {X 0,Y 383.253,Z 378.744,A -85,B 0,C 180,E1 -12068.436,E2 -12068.436} C_VEL
LIN {X 0,Y 383.1,Z 378.761,A -85,B 0,C 180,E1 -12071.642,E2 -12071.642} C_VEL
LIN {X 0,Y 383.104,Z 378.765,A -85,B 0,C 180,E1 -12074.882,E2 -12074.882} C_VEL
LIN {X 0,Y 383.082,Z 378.764,A -85,B 0,C 180,E1 -12078.173,E2 -12078.173} C_VEL
LIN {X 0,Y 382.99,Z 378.774,A -85,B 0,C 180,E1 -12081.531,E2 -12081.531} C_VEL
LIN {X 0,Y 383.046,Z 378.77,A -85,B 0,C 180,E1 -12084.961,E2 -12084.961} C_VEL
LIN {X 0,Y 383.034,Z 378.775,A -85,B 0,C 180,E1 -12088.493,E2 -12088.493} C_VEL
LIN {X 0,Y 383.003,Z 378.776,A -85,B 0,C 180,E1 -12092.15,E2 -12092.15} C_VEL
LIN {X 0,Y 383.013,Z 378.776,A -85,B 0,C 180,E1 -12094.669,E2 -12094.669} C_VEL
LIN {X 0,Y 382.998,Z 378.775,A -85,B 0,C 180,E1 -12097.905,E2 -12097.905} C_VEL
LIN {X 0,Y 383.042,Z 378.768,A -85,B 0,C 180,E1 -12101.34,E2 -12101.34} C_VEL
LIN {X 0,Y 383.031,Z 378.776,A -85,B 0,C 180,E1 -12104.31,E2 -12104.31} C_VEL
LIN {X 0,Y 383.007,Z 378.772,A -85,B 0,C 180,E1 -12107.241,E2 -12107.241} C_VEL
LIN {X 0,Y 383.014,Z 378.776,A -85,B 0,C 180,E1 -12110.414,E2 -12110.414} C_VEL
LIN {X 0,Y 383.025,Z 378.775,A -85,B 0,C 180,E1 -12114.045,E2 -12114.045} C_VEL
LIN {X 0,Y 382.986,Z 378.776,A -85,B 0,C 180,E1 -12117.579,E2 -12117.579} C_VEL
LIN {X 0,Y 382.992,Z 378.779,A -85,B 0,C 180,E1 -12120.301,E2 -12120.301} C_VEL
LIN {X 0,Y 383.081,Z 378.769,A -85,B 0,C 180,E1 -12124.022,E2 -12124.022} C_VEL
LIN {X 0,Y 383.082,Z 378.974,A -85,B 0,C 180,E1 -12125.981,E2 -12125.981} C_VEL
LIN {X 0,Y 385.348,Z 390.509,A -85,B 0,C 180,E1 -12129.235,E2 -12129.235} C_VEL
LIN {X 0,Y 387.668,Z 399.161,A -85,B 0,C 180,E1 -12129.535,E2 -12129.535} C_VEL
LIN {X 0,Y 390.473,Z 412.843,A -85,B 0,C 180,E1 -12129.954,E2 -12129.954} C_VEL
LIN {X 0,Y 389.431,Z 496.546,A -85,B 0,C 180,E1 -12131.522,E2 -12131.522} C_VEL
LIN {X 0,Y 388.877,Z 510.005,A -85,B 0,C 180,E1 -12131.972,E2 -12131.972} C_VEL
LIN {X 0,Y 388.227,Z 522.786,A -85,B 0,C 180,E1 -12132.621,E2 -12132.621} C_VEL
LIN {X 0,Y 387.48,Z 534.128,A -85,B 0,C 180,E1 -12133.402,E2 -12133.402} C_VEL
LIN {X 0,Y 386.587,Z 546.067,A -85,B 0,C 180,E1 -12134.477,E2 -12134.477} C_VEL
LIN {X 0,Y 385.757,Z 556.216,A -85,B 0,C 180,E1 -12135.628,E2 -12135.628} C_VEL
LIN {X 0,Y 384.913,Z 564.752,A -85,B 0,C 180,E1 -12136.807,E2 -12136.807} C_VEL
LIN {X 0,Y 384.153,Z 572.611,A -85,B 0,C 180,E1 -12138.123,E2 -12138.123} C_VEL
LIN {X 0,Y 383.365,Z 580.292,A -85,B 0,C 180,E1 -12139.704,E2 -12139.704} C_VEL
LIN {X 0,Y 382.632,Z 587.34,A -85,B 0,C 180,E1 -12141.551,E2 -12141.551} C_VEL
LIN {X 0,Y 382.23,Z 592.11,A -85,B 0,C 180,E1 -12143.166,E2 -12143.166} C_VEL
LIN {X 0,Y 381.992,Z 595.619,A -85,B 0,C 180,E1 -12144.722,E2 -12144.722} C_VEL
LIN {X 0,Y 381.801,Z 597.477,A -85,B 0,C 180,E1 -12145.778,E2 -12145.778} C_VEL
LIN {X 0,Y 381.768,Z 598.871,A -85,B 0,C 180,E1 -12146.834,E2 -12146.834} C_VEL
LIN {X 0,Y 381.738,Z 599.862,A -85,B 0,C 180,E1 -12147.89,E2 -12147.89} C_VEL
LIN {X 0,Y 381.658,Z 600.708,A -85,B 0,C 180,E1 -12150,E2 -12150} C_VEL
LIN {X 0,Y 381.68,Z 600.519,A -85,B 0,C 180,E1 -12151.055,E2 -12151.055} C_VEL
LIN {X 0,Y 381.738,Z 599.935,A -85,B 0,C 180,E1 -12152.11,E2 -12152.11} C_VEL
LIN {X 0,Y 381.767,Z 598.972,A -85,B 0,C 180,E1 -12153.166,E2 -12153.166} C_VEL
LIN {X 0,Y 381.799,Z 597.622,A -85,B 0,C 180,E1 -12154.222,E2 -12154.222} C_VEL
LIN {X 0,Y 382.098,Z 594.759,A -85,B 0,C 180,E1 -12155.806,E2 -12155.806} C_VEL
LIN {X 0,Y 382.354,Z 590.883,A -85,B 0,C 180,E1 -12157.392,E2 -12157.392} C_VEL
LIN {X 0,Y 382.762,Z 585.881,A -85,B 0,C 180,E1 -12158.979,E2 -12158.979} C_VEL
LIN {X 0,Y 383.403,Z 579.578,A -85,B 0,C 180,E1 -12160.562,E2 -12160.562} C_VEL
LIN {X 0,Y 384.223,Z 571.685,A -85,B 0,C 180,E1 -12162.143,E2 -12162.143} C_VEL
LIN {X 0,Y 385.025,Z 563.638,A -85,B 0,C 180,E1 -12163.458,E2 -12163.458} C_VEL
LIN {X 0,Y 385.232,Z 561.909,A -85,B 0,C 180,E1 -12163.712,E2 -12163.712} C_VEL
LIN {X 0,Y 385.028,Z 557.697,A -85,B 0,C 180,E1 -12164.331,E2 -12164.331} C_VEL
LIN {X 0,Y 382.792,Z 550.631,A -85,B 0,C 180,E1 -12165.322,E2 -12165.322} C_VEL
LIN {X 0,Y 380.583,Z 543.06,A -85,B 0,C 180,E1 -12166.226,E2 -12166.226} C_VEL
LIN {X 0,Y 380.407,Z 538.06,A -85,B 0,C 180,E1 -12166.697,E2 -12166.697} C_VEL
LIN {X 0,Y 381.298,Z 526.612,A -85,B 0,C 180,E1 -12167.567,E2 -12167.567} C_VEL
LIN {X 0,Y 382.06,Z 513.934,A -85,B 0,C 180,E1 -12168.292,E2 -12168.292} C_VEL
LIN {X 0,Y 382.595,Z 501.325,A -85,B 0,C 180,E1 -12168.786,E2 -12168.786} C_VEL
LIN {X 0,Y 382.838,Z 483.438,A -85,B 0,C 180,E1 -12169.19,E2 -12169.19} C_VEL
LIN {X 0,Y 383.89,Z 413.956,A -85,B 0,C 180,E1 -12170.49,E2 -12170.49} C_VEL
LIN {X 0,Y 379.864,Z 395.635,A -85,B 0,C 180,E1 -12171.084,E2 -12171.084} C_VEL
LIN {X 0,Y 378.125,Z 390.65,A -85,B 0,C 180,E1 -12171.304,E2 -12171.304} C_VEL
LIN {X 0,Y 376.008,Z 379.654,A -85,B 0,C 180,E1 -12174.5,E2 -12174.5} C_VEL
LIN {X 0,Y 376.02,Z 379.643,A -85,B 0,C 180,E1 -12176.651,E2 -12176.651} C_VEL
LIN {X 0,Y 375.964,Z 379.652,A -85,B 0,C 180,E1 -12180.312,E2 -12180.312} C_VEL
LIN {X 0,Y 375.962,Z 379.654,A -85,B 0,C 180,E1 -12184.11,E2 -12184.11} C_VEL
LIN {X 0,Y 375.953,Z 379.651,A -85,B 0,C 180,E1 -12186.74,E2 -12186.74} C_VEL
LIN {X 0,Y 375.987,Z 379.652,A -85,B 0,C 180,E1 -12189.97,E2 -12189.97} C_VEL
LIN {X 0,Y 375.935,Z 379.66,A -85,B 0,C 180,E1 -12193.764,E2 -12193.764} C_VEL
LIN {X 0,Y 375.985,Z 379.647,A -85,B 0,C 180,E1 -12196.801,E2 -12196.801} C_VEL
LIN {X 0,Y 375.995,Z 379.649,A -85,B 0,C 180,E1 -12200.027,E2 -12200.027} C_VEL
LIN {X 0,Y 375.961,Z 379.655,A -85,B 0,C 180,E1 -12203.494,E2 -12203.494} C_VEL
LIN {X 0,Y 375.955,Z 379.654,A -85,B 0,C 180,E1 -12205.888,E2 -12205.888} C_VEL
LIN {X 0,Y 375.959,Z 379.655,A -85,B 0,C 180,E1 -12209.687,E2 -12209.687} C_VEL
LIN {X 0,Y 375.99,Z 379.647,A -85,B 0,C 180,E1 -12212.141,E2 -12212.141} C_VEL
LIN {X 0,Y 376,Z 379.645,A -85,B 0,C 180,E1 -12214.538,E2 -12214.538} C_VEL
LIN {X 0,Y 375.959,Z 379.651,A -85,B 0,C 180,E1 -12218.045,E2 -12218.045} C_VEL
LIN {X 0,Y 376.017,Z 379.648,A -85,B 0,C 180,E1 -12221.474,E2 -12221.474} C_VEL
LIN {X 0,Y 376.052,Z 379.64,A -85,B 0,C 180,E1 -12224.832,E2 -12224.832} C_VEL
LIN {X 0,Y 376.051,Z 379.639,A -85,B 0,C 180,E1 -12228.137,E2 -12228.137} C_VEL
LIN {X 0,Y 376.25,Z 379.615,A -85,B 0,C 180,E1 -12231.877,E2 -12231.877} C_VEL
LIN {X 0,Y 376.165,Z 379.626,A -85,B 0,C 180,E1 -12234.64,E2 -12234.64} C_VEL
LIN {X 0,Y 376.346,Z 379.602,A -85,B 0,C 180,E1 -12237.86,E2 -12237.86} C_VEL
LIN {X 0,Y 376.483,Z 379.585,A -85,B 0,C 180,E1 -12240,E2 -12240} C_VEL
LIN {X 0,Y 376.185,Z 379.627,A -85,B 0,C 180,E1 -12243.213,E2 -12243.213} C_VEL
LIN {X 0,Y 376.239,Z 379.616,A -85,B 0,C 180,E1 -12246.435,E2 -12246.435} C_VEL
LIN {X 0,Y 376.199,Z 379.623,A -85,B 0,C 180,E1 -12248.595,E2 -12248.595} C_VEL
LIN {X 0,Y 376.051,Z 379.639,A -85,B 0,C 180,E1 -12251.863,E2 -12251.863} C_VEL
LIN {X 0,Y 376.052,Z 379.642,A -85,B 0,C 180,E1 -12255.168,E2 -12255.168} C_VEL
LIN {X 0,Y 376.001,Z 379.648,A -85,B 0,C 180,E1 -12258.527,E2 -12258.527} C_VEL
LIN {X 0,Y 375.957,Z 379.651,A -85,B 0,C 180,E1 -12261.955,E2 -12261.955} C_VEL
LIN {X 0,Y 376,Z 379.646,A -85,B 0,C 180,E1 -12265.462,E2 -12265.462} C_VEL
LIN {X 0,Y 375.964,Z 379.652,A -85,B 0,C 180,E1 -12269.08,E2 -12269.08} C_VEL
LIN {X 0,Y 375.943,Z 379.657,A -85,B 0,C 180,E1 -12272.829,E2 -12272.829} C_VEL
LIN {X 0,Y 375.953,Z 379.651,A -85,B 0,C 180,E1 -12275.416,E2 -12275.416} C_VEL
LIN {X 0,Y 375.973,Z 379.652,A -85,B 0,C 180,E1 -12278.272,E2 -12278.272} C_VEL
LIN {X 0,Y 375.985,Z 379.647,A -85,B 0,C 180,E1 -12281.611,E2 -12281.611} C_VEL
LIN {X 0,Y 375.967,Z 379.649,A -85,B 0,C 180,E1 -12285.263,E2 -12285.263} C_VEL
LIN {X 0,Y 375.948,Z 379.652,A -85,B 0,C 180,E1 -12289.135,E2 -12289.135} C_VEL
LIN {X 0,Y 375.964,Z 379.652,A -85,B 0,C 180,E1 -12291.913,E2 -12291.913} C_VEL
LIN {X 0,Y 375.978,Z 379.648,A -85,B 0,C 180,E1 -12295.333,E2 -12295.333} C_VEL
LIN {X 0,Y 375.958,Z 379.657,A -85,B 0,C 180,E1 -12298.439,E2 -12298.439} C_VEL
LIN {X 0,Y 375.99,Z 379.737,A -85,B 0,C 180,E1 -12300.193,E2 -12300.193} C_VEL
LIN {X 0,Y 378.484,Z 391.089,A -85,B 0,C 180,E1 -12303.038,E2 -12303.038} C_VEL
LIN {X 0,Y 379.885,Z 399.403,A -85,B 0,C 180,E1 -12305.029,E2 -12305.029} C_VEL
LIN {X 0,Y 378.303,Z 416.32,A -85,B 0,C 180,E1 -12308.751,E2 -12308.751} C_VEL
LIN {X 0,Y 382.761,Z 443.663,A -85,B 0,C 180,E1 -12309.544,E2 -12309.544} C_VEL
LIN {X 0,Y 383.513,Z 449.471,A -85,B 0,C 180,E1 -12309.699,E2 -12309.699} C_VEL
LIN {X 0,Y 382.332,Z 524.81,A -85,B 0,C 180,E1 -12311.131,E2 -12311.131} C_VEL
LIN {X 0,Y 381.731,Z 538.032,A -85,B 0,C 180,E1 -12311.588,E2 -12311.588} C_VEL
LIN {X 0,Y 380.9,Z 550.169,A -85,B 0,C 180,E1 -12312.206,E2 -12312.206} C_VEL
LIN {X 0,Y 379.922,Z 562.424,A -85,B 0,C 180,E1 -12313.062,E2 -12313.062} C_VEL
LIN {X 0,Y 378.841,Z 574.019,A -85,B 0,C 180,E1 -12314.12,E2 -12314.12} C_VEL
LIN {X 0,Y 377.835,Z 584.263,A -85,B 0,C 180,E1 -12315.294,E2 -12315.294} C_VEL
LIN {X 0,Y 377.11,Z 593.014,A -85,B 0,C 180,E1 -12316.529,E2 -12316.529} C_VEL
LIN {X 0,Y 376.342,Z 600.901,A -85,B 0,C 180,E1 -12317.873,E2 -12317.873} C_VEL
LIN {X 0,Y 375.551,Z 608.605,A -85,B 0,C 180,E1 -12319.487,E2 -12319.487} C_VEL
LIN {X 0,Y 375.006,Z 615.717,A -85,B 0,C 180,E1 -12321.377,E2 -12321.377} C_VEL
LIN {X 0,Y 374.722,Z 620.451,A -85,B 0,C 180,E1 -12322.998,E2 -12322.998} C_VEL
LIN {X 0,Y 374.55,Z 624.069,A -85,B 0,C 180,E1 -12324.617,E2 -12324.617} C_VEL
LIN {X 0,Y 374.551,Z 625.939,A -85,B 0,C 180,E1 -12325.696,E2 -12325.696} C_VEL
LIN {X 0,Y 374.5,Z 628.338,A -85,B 0,C 180,E1 -12327.849,E2 -12327.849} C_VEL
LIN {X 0,Y 374.584,Z 628.951,A -85,B 0,C 180,E1 -12328.925,E2 -12328.925} C_VEL
LIN {X 0,Y 374.589,Z 629.167,A -85,B 0,C 180,E1 -12330,E2 -12330} C_VEL
LIN {X 0,Y 374.584,Z 628.948,A -85,B 0,C 180,E1 -12331.075,E2 -12331.075} C_VEL
LIN {X 0,Y 374.466,Z 627.33,A -85,B 0,C 180,E1 -12333.228,E2 -12333.228} C_VEL
LIN {X 0,Y 374.552,Z 625.929,A -85,B 0,C 180,E1 -12334.304,E2 -12334.304} C_VEL
LIN {X 0,Y 374.582,Z 622.667,A -85,B 0,C 180,E1 -12336.065,E2 -12336.065} C_VEL
LIN {X 0,Y 374.778,Z 618.987,A -85,B 0,C 180,E1 -12337.543,E2 -12337.543} C_VEL
LIN {X 0,Y 375.197,Z 612.855,A -85,B 0,C 180,E1 -12339.433,E2 -12339.433} C_VEL
LIN {X 0,Y 375.737,Z 606.159,A -85,B 0,C 180,E1 -12341.053,E2 -12341.053} C_VEL
LIN {X 0,Y 376.631,Z 597.862,A -85,B 0,C 180,E1 -12342.665,E2 -12342.665} C_VEL
LIN {X 0,Y 377.437,Z 589.354,A -85,B 0,C 180,E1 -12344.008,E2 -12344.008} C_VEL
LIN {X 0,Y 378.371,Z 578.844,A -85,B 0,C 180,E1 -12345.348,E2 -12345.348} C_VEL
LIN {X 0,Y 379.532,Z 567.025,A -85,B 0,C 180,E1 -12346.541,E2 -12346.541} C_VEL
LIN {X 0,Y 380.521,Z 555.134,A -85,B 0,C 180,E1 -12347.465,E2 -12347.465} C_VEL
LIN {X 0,Y 381.379,Z 542.764,A -85,B 0,C 180,E1 -12348.187,E2 -12348.187} C_VEL
LIN {X 0,Y 382.133,Z 530.059,A -85,B 0,C 180,E1 -12348.705,E2 -12348.705} C_VEL
LIN {X 0,Y 382.479,Z 516.714,A -85,B 0,C 180,E1 -12349.035,E2 -12349.035} C_VEL
LIN {X 0,Y 383.412,Z 448.128,A -85,B 0,C 180,E1 -12350.322,E2 -12350.322} C_VEL
LIN {X 0,Y 378.518,Z 417.894,A -85,B 0,C 180,E1 -12351.192,E2 -12351.192} C_VEL
LIN {X 0,Y 378.286,Z 416.324,A -85,B 0,C 180,E1 -12351.24,E2 -12351.24} C_VEL
LIN {X 0,Y 379.807,Z 400.122,A -85,B 0,C 180,E1 -12354.797,E2 -12354.797} C_VEL
LIN {X 0,Y 379.385,Z 395.804,A -85,B 0,C 180,E1 -12355.806,E2 -12355.806} C_VEL
LIN {X 0,Y 376.919,Z 383.657,A -85,B 0,C 180,E1 -12358.793,E2 -12358.793} C_VEL
LIN {X 0,Y 375.994,Z 379.653,A -85,B 0,C 180,E1 -12359.845,E2 -12359.845} C_VEL
LIN {X 0,Y 375.948,Z 379.656,A -85,B 0,C 180,E1 -12362.828,E2 -12362.828} C_VEL
LIN {X 0,Y 375.956,Z 379.654,A -85,B 0,C 180,E1 -12365.415,E2 -12365.415} C_VEL
LIN {X 0,Y 375.974,Z 379.649,A -85,B 0,C 180,E1 -12368.27,E2 -12368.27} C_VEL
LIN {X 0,Y 375.942,Z 379.659,A -85,B 0,C 180,E1 -12371.602,E2 -12371.602} C_VEL
LIN {X 0,Y 375.976,Z 379.652,A -85,B 0,C 180,E1 -12375.26,E2 -12375.26} C_VEL
LIN {X 0,Y 375.985,Z 379.647,A -85,B 0,C 180,E1 -12378.389,E2 -12378.389} C_VEL
LIN {X 0,Y 375.963,Z 379.652,A -85,B 0,C 180,E1 -12381.911,E2 -12381.911} C_VEL
LIN {X 0,Y 375.974,Z 379.654,A -85,B 0,C 180,E1 -12385.332,E2 -12385.332} C_VEL
LIN {X 0,Y 375.954,Z 379.651,A -85,B 0,C 180,E1 -12388.438,E2 -12388.438} C_VEL
LIN {X 0,Y 375.996,Z 379.646,A -85,B 0,C 180,E1 -12392.141,E2 -12392.141} C_VEL
LIN {X 0,Y 376,Z 379.646,A -85,B 0,C 180,E1 -12394.538,E2 -12394.538} C_VEL
LIN {X 0,Y 375.957,Z 379.651,A -85,B 0,C 180,E1 -12398.045,E2 -12398.045} C_VEL
LIN {X 0,Y 376.001,Z 379.648,A -85,B 0,C 180,E1 -12401.473,E2 -12401.473} C_VEL
LIN {X 0,Y 376.052,Z 379.642,A -85,B 0,C 180,E1 -12404.832,E2 -12404.832} C_VEL
LIN {X 0,Y 376.051,Z 379.639,A -85,B 0,C 180,E1 -12408.137,E2 -12408.137} C_VEL
LIN {X 0,Y 376.25,Z 379.614,A -85,B 0,C 180,E1 -12411.877,E2 -12411.877} C_VEL
LIN {X 0,Y 376.165,Z 379.627,A -85,B 0,C 180,E1 -12414.64,E2 -12414.64} C_VEL
LIN {X 0,Y 376.346,Z 379.602,A -85,B 0,C 180,E1 -12417.86,E2 -12417.86} C_VEL
LIN {X 0,Y 376.483,Z 379.585,A -85,B 0,C 180,E1 -12420,E2 -12420} C_VEL
LIN {X 0,Y 376.184,Z 379.625,A -85,B 0,C 180,E1 -12423.213,E2 -12423.213} C_VEL
LIN {X 0,Y 376.226,Z 379.618,A -85,B 0,C 180,E1 -12426.645,E2 -12426.645} C_VEL
LIN {X 0,Y 376.199,Z 379.624,A -85,B 0,C 180,E1 -12428.595,E2 -12428.595} C_VEL
LIN {X 0,Y 376.051,Z 379.639,A -85,B 0,C 180,E1 -12431.863,E2 -12431.863} C_VEL
LIN {X 0,Y 376.052,Z 379.641,A -85,B 0,C 180,E1 -12435.168,E2 -12435.168} C_VEL
LIN {X 0,Y 376.017,Z 379.648,A -85,B 0,C 180,E1 -12438.526,E2 -12438.526} C_VEL
LIN {X 0,Y 375.959,Z 379.651,A -85,B 0,C 180,E1 -12441.955,E2 -12441.955} C_VEL
LIN {X 0,Y 376,Z 379.645,A -85,B 0,C 180,E1 -12445.462,E2 -12445.462} C_VEL
LIN {X 0,Y 375.964,Z 379.651,A -85,B 0,C 180,E1 -12449.08,E2 -12449.08} C_VEL
LIN {X 0,Y 375.944,Z 379.655,A -85,B 0,C 180,E1 -12452.829,E2 -12452.829} C_VEL
LIN {X 0,Y 375.953,Z 379.651,A -85,B 0,C 180,E1 -12455.416,E2 -12455.416} C_VEL
LIN {X 0,Y 375.973,Z 379.653,A -85,B 0,C 180,E1 -12458.272,E2 -12458.272} C_VEL
LIN {X 0,Y 375.986,Z 379.647,A -85,B 0,C 180,E1 -12461.611,E2 -12461.611} C_VEL
LIN {X 0,Y 375.966,Z 379.649,A -85,B 0,C 180,E1 -12465.263,E2 -12465.263} C_VEL
LIN {X 0,Y 375.938,Z 379.653,A -85,B 0,C 180,E1 -12469.134,E2 -12469.134} C_VEL
LIN {X 0,Y 375.965,Z 379.653,A -85,B 0,C 180,E1 -12471.913,E2 -12471.913} C_VEL
LIN {X 0,Y 375.979,Z 379.648,A -85,B 0,C 180,E1 -12475.333,E2 -12475.333} C_VEL
LIN {X 0,Y 375.957,Z 379.654,A -85,B 0,C 180,E1 -12478.439,E2 -12478.439} C_VEL
LIN {X 0,Y 375.984,Z 379.653,A -85,B 0,C 180,E1 -12482.141,E2 -12482.141} C_VEL
LIN {X 0,Y 376.015,Z 379.65,A -85,B 0,C 180,E1 -12485.132,E2 -12485.132} C_VEL
LIN {X 0,Y 376.015,Z 379.747,A -85,B 0,C 180,E1 -12485.647,E2 -12485.647} C_VEL
LIN {X 0,Y 378.204,Z 390.72,A -85,B 0,C 180,E1 -12488.822,E2 -12488.822} C_VEL
LIN {X 0,Y 380.828,Z 399.384,A -85,B 0,C 180,E1 -12489.149,E2 -12489.149} C_VEL
LIN {X 0,Y 383.915,Z 414.598,A -85,B 0,C 180,E1 -12489.625,E2 -12489.625} C_VEL
LIN {X 0,Y 382.634,Z 498.008,A -85,B 0,C 180,E1 -12491.216,E2 -12491.216} C_VEL
LIN {X 0,Y 382.05,Z 511.803,A -85,B 0,C 180,E1 -12491.708,E2 -12491.708} C_VEL
LIN {X 0,Y 381.408,Z 524.16,A -85,B 0,C 180,E1 -12492.369,E2 -12492.369} C_VEL
LIN {X 0,Y 380.595,Z 535.984,A -85,B 0,C 180,E1 -12493.231,E2 -12493.231} C_VEL
LIN {X 0,Y 379.699,Z 546.99,A -85,B 0,C 180,E1 -12494.258,E2 -12494.258} C_VEL
LIN {X 0,Y 378.798,Z 557.545,A -85,B 0,C 180,E1 -12495.495,E2 -12495.495} C_VEL
LIN {X 0,Y 377.841,Z 566.714,A -85,B 0,C 180,E1 -12496.83,E2 -12496.83} C_VEL
LIN {X 0,Y 376.861,Z 575.616,A -85,B 0,C 180,E1 -12498.436,E2 -12498.436} C_VEL
LIN {X 0,Y 376.122,Z 582.778,A -85,B 0,C 180,E1 -12500.047,E2 -12500.047} C_VEL
LIN {X 0,Y 375.598,Z 587.609,A -85,B 0,C 180,E1 -12501.391,E2 -12501.391} C_VEL
LIN {X 0,Y 375.149,Z 592.726,A -85,B 0,C 180,E1 -12503.169,E2 -12503.169} C_VEL
LIN {X 0,Y 374.946,Z 595.887,A -85,B 0,C 180,E1 -12504.622,E2 -12504.622} C_VEL
LIN {X 0,Y 374.731,Z 597.744,A -85,B 0,C 180,E1 -12505.698,E2 -12505.698} C_VEL
LIN {X 0,Y 374.676,Z 599.139,A -85,B 0,C 180,E1 -12506.774,E2 -12506.774} C_VEL
LIN {X 0,Y 374.644,Z 600.13,A -85,B 0,C 180,E1 -12507.85,E2 -12507.85} C_VEL
LIN {X 0,Y 374.591,Z 600.974,A -85,B 0,C 180,E1 -12510,E2 -12510} C_VEL
LIN {X 0,Y 374.597,Z 600.785,A -85,B 0,C 180,E1 -12511.075,E2 -12511.075} C_VEL
LIN {X 0,Y 374.644,Z 600.202,A -85,B 0,C 180,E1 -12512.15,E2 -12512.15} C_VEL
LIN {X 0,Y 374.729,Z 597.888,A -85,B 0,C 180,E1 -12514.302,E2 -12514.302} C_VEL
LIN {X 0,Y 375.039,Z 595.025,A -85,B 0,C 180,E1 -12515.916,E2 -12515.916} C_VEL
LIN {X 0,Y 375.306,Z 591.15,A -85,B 0,C 180,E1 -12517.532,E2 -12517.532} C_VEL
LIN {X 0,Y 375.757,Z 586.146,A -85,B 0,C 180,E1 -12519.148,E2 -12519.148} C_VEL
LIN {X 0,Y 376.432,Z 579.842,A -85,B 0,C 180,E1 -12520.76,E2 -12520.76} C_VEL
LIN {X 0,Y 377.255,Z 571.95,A -85,B 0,C 180,E1 -12522.37,E2 -12522.37} C_VEL
LIN {X 0,Y 378.315,Z 562.467,A -85,B 0,C 180,E1 -12523.922,E2 -12523.922} C_VEL
LIN {X 0,Y 379.22,Z 552.857,A -85,B 0,C 180,E1 -12525.19,E2 -12525.19} C_VEL
LIN {X 0,Y 380.083,Z 541.608,A -85,B 0,C 180,E1 -12526.378,E2 -12526.378} C_VEL
LIN {X 0,Y 380.407,Z 538.06,A -85,B 0,C 180,E1 -12526.697,E2 -12526.697} C_VEL
LIN {X 0,Y 380.333,Z 532.961,A -85,B 0,C 180,E1 -12527.137,E2 -12527.137} C_VEL
LIN {X 0,Y 378.331,Z 524.504,A -85,B 0,C 180,E1 -12527.866,E2 -12527.866} C_VEL
LIN {X 0,Y 376.03,Z 515.823,A -85,B 0,C 180,E1 -12528.508,E2 -12528.508} C_VEL
LIN {X 0,Y 375.508,Z 510.275,A -85,B 0,C 180,E1 -12528.809,E2 -12528.809} C_VEL
LIN {X 0,Y 375.996,Z 496.966,A -85,B 0,C 180,E1 -12529.27,E2 -12529.27} C_VEL
LIN {X 0,Y 377.278,Z 415.05,A -85,B 0,C 180,E1 -12530.849,E2 -12530.849} C_VEL
LIN {X 0,Y 373.497,Z 397.977,A -85,B 0,C 180,E1 -12531.419,E2 -12531.419} C_VEL
LIN {X 0,Y 370.984,Z 390.914,A -85,B 0,C 180,E1 -12531.737,E2 -12531.737} C_VEL
LIN {X 0,Y 368.973,Z 380.529,A -85,B 0,C 180,E1 -12534.849,E2 -12534.849} C_VEL
LIN {X 0,Y 368.963,Z 380.524,A -85,B 0,C 180,E1 -12538.437,E2 -12538.437} C_VEL
LIN {X 0,Y 368.898,Z 380.533,A -85,B 0,C 180,E1 -12542.237,E2 -12542.237} C_VEL
LIN {X 0,Y 368.928,Z 380.526,A -85,B 0,C 180,E1 -12545.001,E2 -12545.001} C_VEL
LIN {X 0,Y 368.908,Z 380.529,A -85,B 0,C 180,E1 -12548.64,E2 -12548.64} C_VEL
LIN {X 0,Y 368.879,Z 380.536,A -85,B 0,C 180,E1 -12552.009,E2 -12552.009} C_VEL
LIN {X 0,Y 368.951,Z 380.525,A -85,B 0,C 180,E1 -12555.186,E2 -12555.186} C_VEL
LIN {X 0,Y 368.942,Z 380.526,A -85,B 0,C 180,E1 -12558.186,E2 -12558.186} C_VEL
LIN {X 0,Y 368.909,Z 380.532,A -85,B 0,C 180,E1 -12561.358,E2 -12561.358} C_VEL
LIN {X 0,Y 368.932,Z 380.528,A -85,B 0,C 180,E1 -12565.146,E2 -12565.146} C_VEL
LIN {X 0,Y 368.924,Z 380.528,A -85,B 0,C 180,E1 -12569.046,E2 -12569.046} C_VEL
LIN {X 0,Y 368.974,Z 380.526,A -85,B 0,C 180,E1 -12571.563,E2 -12571.563} C_VEL
LIN {X 0,Y 368.994,Z 380.519,A -85,B 0,C 180,E1 -12574.019,E2 -12574.019} C_VEL
LIN {X 0,Y 368.927,Z 380.531,A -85,B 0,C 180,E1 -12577.604,E2 -12577.604} C_VEL
LIN {X 0,Y 368.976,Z 380.524,A -85,B 0,C 180,E1 -12581.107,E2 -12581.107} C_VEL
LIN {X 0,Y 368.991,Z 380.518,A -85,B 0,C 180,E1 -12584.535,E2 -12584.535} C_VEL
LIN {X 0,Y 369.005,Z 380.517,A -85,B 0,C 180,E1 -12587.907,E2 -12587.907} C_VEL
LIN {X 0,Y 369.221,Z 380.491,A -85,B 0,C 180,E1 -12591.801,E2 -12591.801} C_VEL
LIN {X 0,Y 369.137,Z 380.501,A -85,B 0,C 180,E1 -12594.537,E2 -12594.537} C_VEL
LIN {X 0,Y 369.311,Z 380.479,A -85,B 0,C 180,E1 -12597.819,E2 -12597.819} C_VEL
LIN {X 0,Y 369.452,Z 380.461,A -85,B 0,C 180,E1 -12600,E2 -12600} C_VEL
LIN {X 0,Y 369.312,Z 380.478,A -85,B 0,C 180,E1 -12602.181,E2 -12602.181} C_VEL
LIN {X 0,Y 369.201,Z 380.494,A -85,B 0,C 180,E1 -12606.558,E2 -12606.558} C_VEL
LIN {X 0,Y 369.132,Z 380.505,A -85,B 0,C 180,E1 -12608.761,E2 -12608.761} C_VEL
LIN {X 0,Y 369.005,Z 380.517,A -85,B 0,C 180,E1 -12612.093,E2 -12612.093} C_VEL
LIN {X 0,Y 368.991,Z 380.519,A -85,B 0,C 180,E1 -12615.465,E2 -12615.465} C_VEL
LIN {X 0,Y 368.951,Z 380.529,A -85,B 0,C 180,E1 -12618.895,E2 -12618.895} C_VEL
LIN {X 0,Y 368.926,Z 380.529,A -85,B 0,C 180,E1 -12622.396,E2 -12622.396} C_VEL
LIN {X 0,Y 368.993,Z 380.518,A -85,B 0,C 180,E1 -12625.981,E2 -12625.981} C_VEL
LIN {X 0,Y 368.955,Z 380.528,A -85,B 0,C 180,E1 -12628.812,E2 -12628.812} C_VEL
LIN {X 0,Y 368.892,Z 380.533,A -85,B 0,C 180,E1 -12632.239,E2 -12632.239} C_VEL
LIN {X 0,Y 368.924,Z 380.529,A -85,B 0,C 180,E1 -12635.002,E2 -12635.002} C_VEL
LIN {X 0,Y 368.909,Z 380.534,A -85,B 0,C 180,E1 -12638.642,E2 -12638.642} C_VEL
LIN {X 0,Y 368.938,Z 380.527,A -85,B 0,C 180,E1 -12642.021,E2 -12642.021} C_VEL
LIN {X 0,Y 368.921,Z 380.527,A -85,B 0,C 180,E1 -12645.183,E2 -12645.183} C_VEL
LIN {X 0,Y 368.888,Z 380.535,A -85,B 0,C 180,E1 -12648.18,E2 -12648.18} C_VEL
LIN {X 0,Y 368.908,Z 380.528,A -85,B 0,C 180,E1 -12651.36,E2 -12651.36} C_VEL
LIN {X 0,Y 368.935,Z 380.525,A -85,B 0,C 180,E1 -12655.147,E2 -12655.147} C_VEL
LIN {X 0,Y 368.928,Z 380.531,A -85,B 0,C 180,E1 -12659.047,E2 -12659.047} C_VEL
LIN {X 0,Y 368.954,Z 380.624,A -85,B 0,C 180,E1 -12659.842,E2 -12659.842} C_VEL
LIN {X 0,Y 371.656,Z 392.997,A -85,B 0,C 180,E1 -12663.01,E2 -12663.01} C_VEL
LIN {X 0,Y 372.925,Z 400.17,A -85,B 0,C 180,E1 -12664.768,E2 -12664.768} C_VEL
LIN {X 0,Y 371.844,Z 412.293,A -85,B 0,C 180,E1 -12667.497,E2 -12667.497} C_VEL
LIN {X 0,Y 371.427,Z 415.953,A -85,B 0,C 180,E1 -12668.316,E2 -12668.316} C_VEL
LIN {X 0,Y 375.398,Z 439.786,A -85,B 0,C 180,E1 -12669.052,E2 -12669.052} C_VEL
LIN {X 0,Y 376.845,Z 450.386,A -85,B 0,C 180,E1 -12669.347,E2 -12669.347} C_VEL
LIN {X 0,Y 375.642,Z 524.556,A -85,B 0,C 180,E1 -12670.782,E2 -12670.782} C_VEL
LIN {X 0,Y 375.004,Z 537.773,A -85,B 0,C 180,E1 -12671.245,E2 -12671.245} C_VEL
LIN {X 0,Y 374.142,Z 549.909,A -85,B 0,C 180,E1 -12671.874,E2 -12671.874} C_VEL
LIN {X 0,Y 373.13,Z 562.161,A -85,B 0,C 180,E1 -12672.744,E2 -12672.744} C_VEL
LIN {X 0,Y 372.001,Z 573.755,A -85,B 0,C 180,E1 -12673.82,E2 -12673.82} C_VEL
LIN {X 0,Y 370.85,Z 584.896,A -85,B 0,C 180,E1 -12675.129,E2 -12675.129} C_VEL
LIN {X 0,Y 370.017,Z 594.427,A -85,B 0,C 180,E1 -12676.546,E2 -12676.546} C_VEL
LIN {X 0,Y 369.02,Z 603.374,A -85,B 0,C 180,E1 -12678.186,E2 -12678.186} C_VEL
LIN {X 0,Y 368.332,Z 610.581,A -85,B 0,C 180,E1 -12679.835,E2 -12679.835} C_VEL
LIN {X 0,Y 367.838,Z 617.15,A -85,B 0,C 180,E1 -12681.762,E2 -12681.762} C_VEL
LIN {X 0,Y 367.563,Z 621.499,A -85,B 0,C 180,E1 -12683.413,E2 -12683.413} C_VEL
LIN {X 0,Y 367.464,Z 623.802,A -85,B 0,C 180,E1 -12684.513,E2 -12684.513} C_VEL
LIN {X 0,Y 367.456,Z 625.671,A -85,B 0,C 180,E1 -12685.612,E2 -12685.612} C_VEL
LIN {X 0,Y 367.399,Z 628.071,A -85,B 0,C 180,E1 -12687.807,E2 -12687.807} C_VEL
LIN {X 0,Y 367.484,Z 628.684,A -85,B 0,C 180,E1 -12688.904,E2 -12688.904} C_VEL
LIN {X 0,Y 367.505,Z 628.9,A -85,B 0,C 180,E1 -12690,E2 -12690} C_VEL
LIN {X 0,Y 367.484,Z 628.68,A -85,B 0,C 180,E1 -12691.096,E2 -12691.096} C_VEL
LIN {X 0,Y 367.384,Z 627.063,A -85,B 0,C 180,E1 -12693.29,E2 -12693.29} C_VEL
LIN {X 0,Y 367.457,Z 625.66,A -85,B 0,C 180,E1 -12694.388,E2 -12694.388} C_VEL
LIN {X 0,Y 367.479,Z 622.756,A -85,B 0,C 180,E1 -12696.013,E2 -12696.013} C_VEL
LIN {X 0,Y 367.707,Z 618.717,A -85,B 0,C 180,E1 -12697.689,E2 -12697.689} C_VEL
LIN {X 0,Y 368.157,Z 612.585,A -85,B 0,C 180,E1 -12699.615,E2 -12699.615} C_VEL
LIN {X 0,Y 368.746,Z 605.889,A -85,B 0,C 180,E1 -12701.265,E2 -12701.265} C_VEL
LIN {X 0,Y 369.686,Z 597.591,A -85,B 0,C 180,E1 -12702.907,E2 -12702.907} C_VEL
LIN {X 0,Y 370.541,Z 589.084,A -85,B 0,C 180,E1 -12704.274,E2 -12704.274} C_VEL
LIN {X 0,Y 371.499,Z 578.572,A -85,B 0,C 180,E1 -12705.639,E2 -12705.639} C_VEL
LIN {X 0,Y 372.705,Z 566.753,A -85,B 0,C 180,E1 -12706.853,E2 -12706.853} C_VEL
LIN {X 0,Y 373.734,Z 554.861,A -85,B 0,C 180,E1 -12707.793,E2 -12707.793} C_VEL
LIN {X 0,Y 374.642,Z 542.49,A -85,B 0,C 180,E1 -12708.526,E2 -12708.526} C_VEL
LIN {X 0,Y 375.428,Z 529.781,A -85,B 0,C 180,E1 -12709.052,E2 -12709.052} C_VEL
LIN {X 0,Y 375.785,Z 516.427,A -85,B 0,C 180,E1 -12709.388,E2 -12709.388} C_VEL
LIN {X 0,Y 376.681,Z 448.551,A -85,B 0,C 180,E1 -12710.687,E2 -12710.687} C_VEL
LIN {X 0,Y 372.002,Z 419.418,A -85,B 0,C 180,E1 -12711.545,E2 -12711.545} C_VEL
LIN {X 0,Y 371.438,Z 416.057,A -85,B 0,C 180,E1 -12711.65,E2 -12711.65} C_VEL
LIN {X 0,Y 372.863,Z 401.691,A -85,B 0,C 180,E1 -12714.867,E2 -12714.867} C_VEL
LIN {X 0,Y 372.609,Z 398.127,A -85,B 0,C 180,E1 -12715.709,E2 -12715.709} C_VEL
LIN {X 0,Y 370.338,Z 386.616,A -85,B 0,C 180,E1 -12718.586,E2 -12718.586} C_VEL
LIN {X 0,Y 368.955,Z 380.529,A -85,B 0,C 180,E1 -12720.198,E2 -12720.198} C_VEL
LIN {X 0,Y 368.895,Z 380.536,A -85,B 0,C 180,E1 -12723.537,E2 -12723.537} C_VEL
LIN {X 0,Y 368.901,Z 380.53,A -85,B 0,C 180,E1 -12726.855,E2 -12726.855} C_VEL
LIN {X 0,Y 368.932,Z 380.526,A -85,B 0,C 180,E1 -12730.366,E2 -12730.366} C_VEL
LIN {X 0,Y 368.887,Z 380.537,A -85,B 0,C 180,E1 -12733.616,E2 -12733.616} C_VEL
LIN {X 0,Y 368.935,Z 380.525,A -85,B 0,C 180,E1 -12736.703,E2 -12736.703} C_VEL
LIN {X 0,Y 368.949,Z 380.528,A -85,B 0,C 180,E1 -12739.635,E2 -12739.635} C_VEL
LIN {X 0,Y 368.898,Z 380.533,A -85,B 0,C 180,E1 -12743.143,E2 -12743.143} C_VEL
LIN {X 0,Y 368.891,Z 380.531,A -85,B 0,C 180,E1 -12746.461,E2 -12746.461} C_VEL
LIN {X 0,Y 368.917,Z 380.527,A -85,B 0,C 180,E1 -12750.31,E2 -12750.31} C_VEL
LIN {X 0,Y 368.975,Z 380.524,A -85,B 0,C 180,E1 -12753.535,E2 -12753.535} C_VEL
LIN {X 0,Y 368.96,Z 380.522,A -85,B 0,C 180,E1 -12756.421,E2 -12756.421} C_VEL
LIN {X 0,Y 368.929,Z 380.526,A -85,B 0,C 180,E1 -12759.947,E2 -12759.947} C_VEL
LIN {X 0,Y 368.969,Z 380.525,A -85,B 0,C 180,E1 -12763.398,E2 -12763.398} C_VEL
LIN {X 0,Y 369.052,Z 380.514,A -85,B 0,C 180,E1 -12766.79,E2 -12766.79} C_VEL
LIN {X 0,Y 369.065,Z 380.509,A -85,B 0,C 180,E1 -12770.132,E2 -12770.132} C_VEL
LIN {X 0,Y 369.18,Z 380.495,A -85,B 0,C 180,E1 -12772.342,E2 -12772.342} C_VEL
LIN {X 0,Y 369.137,Z 380.502,A -85,B 0,C 180,E1 -12774.537,E2 -12774.537} C_VEL
LIN {X 0,Y 369.311,Z 380.478,A -85,B 0,C 180,E1 -12777.819,E2 -12777.819} C_VEL
LIN {X 0,Y 369.452,Z 380.461,A -85,B 0,C 180,E1 -12780,E2 -12780} C_VEL
LIN {X 0,Y 369.312,Z 380.479,A -85,B 0,C 180,E1 -12782.181,E2 -12782.181} C_VEL
LIN {X 0,Y 369.195,Z 380.495,A -85,B 0,C 180,E1 -12786.633,E2 -12786.633} C_VEL
LIN {X 0,Y 369.132,Z 380.507,A -85,B 0,C 180,E1 -12788.761,E2 -12788.761} C_VEL
LIN {X 0,Y 369.005,Z 380.517,A -85,B 0,C 180,E1 -12792.093,E2 -12792.093} C_VEL
LIN {X 0,Y 368.991,Z 380.519,A -85,B 0,C 180,E1 -12795.465,E2 -12795.465} C_VEL
LIN {X 0,Y 368.976,Z 380.524,A -85,B 0,C 180,E1 -12798.893,E2 -12798.893} C_VEL
LIN {X 0,Y 368.927,Z 380.53,A -85,B 0,C 180,E1 -12802.396,E2 -12802.396} C_VEL
LIN {X 0,Y 368.994,Z 380.519,A -85,B 0,C 180,E1 -12805.981,E2 -12805.981} C_VEL
LIN {X 0,Y 368.955,Z 380.526,A -85,B 0,C 180,E1 -12808.812,E2 -12808.812} C_VEL
LIN {X 0,Y 368.892,Z 380.534,A -85,B 0,C 180,E1 -12812.239,E2 -12812.239} C_VEL
LIN {X 0,Y 368.924,Z 380.528,A -85,B 0,C 180,E1 -12815.002,E2 -12815.002} C_VEL
LIN {X 0,Y 368.909,Z 380.533,A -85,B 0,C 180,E1 -12818.642,E2 -12818.642} C_VEL
LIN {X 0,Y 368.948,Z 380.526,A -85,B 0,C 180,E1 -12822.022,E2 -12822.022} C_VEL
LIN {X 0,Y 368.92,Z 380.527,A -85,B 0,C 180,E1 -12825.183,E2 -12825.183} C_VEL
LIN {X 0,Y 368.881,Z 380.537,A -85,B 0,C 180,E1 -12828.179,E2 -12828.179} C_VEL
LIN {X 0,Y 368.908,Z 380.529,A -85,B 0,C 180,E1 -12831.36,E2 -12831.36} C_VEL
LIN {X 0,Y 368.936,Z 380.525,A -85,B 0,C 180,E1 -12835.147,E2 -12835.147} C_VEL
LIN {X 0,Y 368.929,Z 380.526,A -85,B 0,C 180,E1 -12839.047,E2 -12839.047} C_VEL
LIN {X 0,Y 368.963,Z 380.522,A -85,B 0,C 180,E1 -12842.797,E2 -12842.797} C_VEL
LIN {X 0,Y 369.01,Z 380.664,A -85,B 0,C 180,E1 -12845.34,E2 -12845.34} C_VEL
LIN {X 0,Y 371.062,Z 391.026,A -85,B 0,C 180,E1 -12848.394,E2 -12848.394} C_VEL
LIN {X 0,Y 374.301,Z 400.8,A -85,B 0,C 180,E1 -12848.79,E2 -12848.79} C_VEL
LIN {X 0,Y 377.226,Z 415.119,A -85,B 0,C 180,E1 -12849.252,E2 -12849.252} C_VEL
LIN {X 0,Y 375.947,Z 498.29,A -85,B 0,C 180,E1 -12850.869,E2 -12850.869} C_VEL
LIN {X 0,Y 375.342,Z 512.08,A -85,B 0,C 180,E1 -12851.369,E2 -12851.369} C_VEL
LIN {X 0,Y 374.664,Z 524.434,A -85,B 0,C 180,E1 -12852.041,E2 -12852.041} C_VEL
LIN {X 0,Y 373.818,Z 536.257,A -85,B 0,C 180,E1 -12852.917,E2 -12852.917} C_VEL
LIN {X 0,Y 372.819,Z 547.899,A -85,B 0,C 180,E1 -12854.03,E2 -12854.03} C_VEL
LIN {X 0,Y 371.937,Z 557.815,A -85,B 0,C 180,E1 -12855.221,E2 -12855.221} C_VEL
LIN {X 0,Y 370.947,Z 566.983,A -85,B 0,C 180,E1 -12856.58,E2 -12856.58} C_VEL
LIN {X 0,Y 369.919,Z 575.885,A -85,B 0,C 180,E1 -12858.215,E2 -12858.215} C_VEL
LIN {X 0,Y 369.128,Z 583.048,A -85,B 0,C 180,E1 -12859.857,E2 -12859.857} C_VEL
LIN {X 0,Y 368.582,Z 587.878,A -85,B 0,C 180,E1 -12861.226,E2 -12861.226} C_VEL
LIN {X 0,Y 368.093,Z 593.245,A -85,B 0,C 180,E1 -12863.14,E2 -12863.14} C_VEL
LIN {X 0,Y 367.901,Z 596.154,A -85,B 0,C 180,E1 -12864.519,E2 -12864.519} C_VEL
LIN {X 0,Y 367.666,Z 598.012,A -85,B 0,C 180,E1 -12865.615,E2 -12865.615} C_VEL
LIN {X 0,Y 367.585,Z 599.406,A -85,B 0,C 180,E1 -12866.712,E2 -12866.712} C_VEL
LIN {X 0,Y 367.55,Z 600.397,A -85,B 0,C 180,E1 -12867.808,E2 -12867.808} C_VEL
LIN {X 0,Y 367.507,Z 601.24,A -85,B 0,C 180,E1 -12870,E2 -12870} C_VEL
LIN {X 0,Y 367.516,Z 601.051,A -85,B 0,C 180,E1 -12871.096,E2 -12871.096} C_VEL
LIN {X 0,Y 367.55,Z 600.468,A -85,B 0,C 180,E1 -12872.192,E2 -12872.192} C_VEL
LIN {X 0,Y 367.664,Z 598.154,A -85,B 0,C 180,E1 -12874.385,E2 -12874.385} C_VEL
LIN {X 0,Y 367.984,Z 595.291,A -85,B 0,C 180,E1 -12876.029,E2 -12876.029} C_VEL
LIN {X 0,Y 368.268,Z 591.416,A -85,B 0,C 180,E1 -12877.677,E2 -12877.677} C_VEL
LIN {X 0,Y 368.74,Z 586.412,A -85,B 0,C 180,E1 -12879.323,E2 -12879.323} C_VEL
LIN {X 0,Y 369.453,Z 580.108,A -85,B 0,C 180,E1 -12880.966,E2 -12880.966} C_VEL
LIN {X 0,Y 370.321,Z 572.215,A -85,B 0,C 180,E1 -12882.606,E2 -12882.606} C_VEL
LIN {X 0,Y 371.267,Z 564.164,A -85,B 0,C 180,E1 -12883.966,E2 -12883.966} C_VEL
LIN {X 0,Y 372.277,Z 554.34,A -85,B 0,C 180,E1 -12885.325,E2 -12885.325} C_VEL
LIN {X 0,Y 373.104,Z 544.673,A -85,B 0,C 180,E1 -12886.412,E2 -12886.412} C_VEL
LIN {X 0,Y 374.029,Z 534.202,A -85,B 0,C 180,E1 -12887.355,E2 -12887.355} C_VEL
LIN {X 0,Y 374.927,Z 521.589,A -85,B 0,C 180,E1 -12888.228,E2 -12888.228} C_VEL
LIN {X 0,Y 375.508,Z 510.275,A -85,B 0,C 180,E1 -12888.809,E2 -12888.809} C_VEL
LIN {X 0,Y 375.042,Z 504.635,A -85,B 0,C 180,E1 -12889.073,E2 -12889.073} C_VEL
LIN {X 0,Y 372.601,Z 495.421,A -85,B 0,C 180,E1 -12889.493,E2 -12889.493} C_VEL
LIN {X 0,Y 370.115,Z 486.1,A -85,B 0,C 180,E1 -12889.836,E2 -12889.836} C_VEL
LIN {X 0,Y 369.596,Z 480.297,A -85,B 0,C 180,E1 -12889.98,E2 -12889.98} C_VEL
LIN {X 0,Y 370.68,Z 416.14,A -85,B 0,C 180,E1 -12891.221,E2 -12891.221} C_VEL
LIN {X 0,Y 367.019,Z 399.861,A -85,B 0,C 180,E1 -12891.782,E2 -12891.782} C_VEL
LIN {X 0,Y 363.836,Z 391.168,A -85,B 0,C 180,E1 -12892.192,E2 -12892.192} C_VEL
LIN {X 0,Y 361.942,Z 381.403,A -85,B 0,C 180,E1 -12895.149,E2 -12895.149} C_VEL
LIN {X 0,Y 361.909,Z 381.405,A -85,B 0,C 180,E1 -12897.778,E2 -12897.778} C_VEL
LIN {X 0,Y 361.837,Z 381.412,A -85,B 0,C 180,E1 -12901.629,E2 -12901.629} C_VEL
LIN {X 0,Y 361.874,Z 381.406,A -85,B 0,C 180,E1 -12905.344,E2 -12905.344} C_VEL
LIN {X 0,Y 361.869,Z 381.406,A -85,B 0,C 180,E1 -12909.026,E2 -12909.026} C_VEL
LIN {X 0,Y 361.836,Z 381.41,A -85,B 0,C 180,E1 -12912.828,E2 -12912.828} C_VEL
LIN {X 0,Y 361.895,Z 381.406,A -85,B 0,C 180,E1 -12915.933,E2 -12915.933} C_VEL
LIN {X 0,Y 361.902,Z 381.403,A -85,B 0,C 180,E1 -12919.231,E2 -12919.231} C_VEL
LIN {X 0,Y 361.865,Z 381.407,A -85,B 0,C 180,E1 -12922.981,E2 -12922.981} C_VEL
LIN {X 0,Y 361.856,Z 381.407,A -85,B 0,C 180,E1 -12926.629,E2 -12926.629} C_VEL
LIN {X 0,Y 361.869,Z 381.41,A -85,B 0,C 180,E1 -12929.671,E2 -12929.671} C_VEL
LIN {X 0,Y 361.948,Z 381.402,A -85,B 0,C 180,E1 -12933.474,E2 -12933.474} C_VEL
LIN {X 0,Y 361.884,Z 381.407,A -85,B 0,C 180,E1 -12937.144,E2 -12937.144} C_VEL
LIN {X 0,Y 361.915,Z 381.401,A -85,B 0,C 180,E1 -12940.724,E2 -12940.724} C_VEL
LIN {X 0,Y 361.939,Z 381.397,A -85,B 0,C 180,E1 -12944.226,E2 -12944.226} C_VEL
LIN {X 0,Y 361.993,Z 381.39,A -85,B 0,C 180,E1 -12946.527,E2 -12946.527} C_VEL
LIN {X 0,Y 362.028,Z 381.386,A -85,B 0,C 180,E1 -12949.938,E2 -12949.938} C_VEL
LIN {X 0,Y 362.143,Z 381.371,A -85,B 0,C 180,E1 -12952.192,E2 -12952.192} C_VEL
